                        IF fb_json.HasMember(json_FeederConfigLeft, 'EmptyDelay') THEN
                            json_value := fb_json.FindMember(json_FeederConfigLeft, 'EmptyDelay');
                            PERS.recipeList[i + 0].st120.FeederConfigLeft.EmptyDelay
                                := TO_DINT(fb_json.GetInt(json_value));
                        END_IF
                    END_IF

                    IF fb_json.HasMember(json_st120, 'FeederConfigRight') THEN
                        json_FeederConfigRight := fb_json.FindMember(json_st120, 'FeederConfigRight');

                        IF fb_json.HasMember(json_FeederConfigRight, 'InFilterDelay') THEN
                            json_value := fb_json.FindMember(json_FeederConfigRight, 'InFilterDelay');
                            PERS.recipeList[i + 0].st120.FeederConfigRight.InFilterDelay
                                := TO_DINT(fb_json.GetInt(json_value));
                        END_IF

                        IF fb_json.HasMember(json_FeederConfigRight, 'StartDelay') THEN
                            json_value := fb_json.FindMember(json_FeederConfigRight, 'StartDelay');
                            PERS.recipeList[i + 0].st120.FeederConfigRight.StartDelay
                                := TO_DINT(fb_json.GetInt(json_value));
                        END_IF

                        IF fb_json.HasMember(json_FeederConfigRight, 'StopDelay') THEN
                            json_value := fb_json.FindMember(json_FeederConfigRight, 'StopDelay');
                            PERS.recipeList[i + 0].st120.FeederConfigRight.StopDelay
                                := TO_DINT(fb_json.GetInt(json_value));
                        END_IF

                        IF fb_json.HasMember(json_FeederConfigRight, 'EmptyDelay') THEN
                            json_value := fb_json.FindMember(json_FeederConfigRight, 'EmptyDelay');
                            PERS.recipeList[i + 0].st120.FeederConfigRight.EmptyDelay
                                := TO_DINT(fb_json.GetInt(json_value));
                        END_IF
                    END_IF
                END_IF

                IF fb_json.HasMember(json_i, 'st125') THEN
                    json_st125 := fb_json.FindMember(json_i, 'st125');

                    IF fb_json.HasMember(json_st125, 'xUseVerLeft') THEN
                        json_value := fb_json.FindMember(json_st125, 'xUseVerLeft');
                        PERS.recipeList[i + 0].st125.xUseVerLeft
                            := (fb_json.GetBool(json_value));
                    END_IF

                    IF fb_json.HasMember(json_st125, 'xUseVerRight') THEN
                        json_value := fb_json.FindMember(json_st125, 'xUseVerRight');
                        PERS.recipeList[i + 0].st125.xUseVerRight
                            := (fb_json.GetBool(json_value));
                    END_IF

                    IF fb_json.HasMember(json_st125, 'FeederConfig') THEN
                        json_FeederConfig := fb_json.FindMember(json_st125, 'FeederConfig');

                        IF fb_json.HasMember(json_FeederConfig, 'InFilterDelay') THEN
                            json_value := fb_json.FindMember(json_FeederConfig, 'InFilterDelay');
                            PERS.recipeList[i + 0].st125.FeederConfig.InFilterDelay
                                := TO_DINT(fb_json.GetInt(json_value));
                        END_IF

                        IF fb_json.HasMember(json_FeederConfig, 'StartDelay') THEN
                            json_value := fb_json.FindMember(json_FeederConfig, 'StartDelay');
                            PERS.recipeList[i + 0].st125.FeederConfig.StartDelay
                                := TO_DINT(fb_json.GetInt(json_value));
                        END_IF

                        IF fb_json.HasMember(json_FeederConfig, 'StopDelay') THEN
                            json_value := fb_json.FindMember(json_FeederConfig, 'StopDelay');
                            PERS.recipeList[i + 0].st125.FeederConfig.StopDelay
                                := TO_DINT(fb_json.GetInt(json_value));
                        END_IF

                        IF fb_json.HasMember(json_FeederConfig, 'EmptyDelay') THEN
                            json_value := fb_json.FindMember(json_FeederConfig, 'EmptyDelay');
                            PERS.recipeList[i + 0].st125.FeederConfig.EmptyDelay
                                := TO_DINT(fb_json.GetInt(json_value));
                        END_IF
                    END_IF
                END_IF

                IF fb_json.HasMember(json_i, 'st145') THEN
                    json_st145 := fb_json.FindMember(json_i, 'st145');

                    IF fb_json.HasMember(json_st145, 'xUseVerLeft') THEN
                        json_value := fb_json.FindMember(json_st145, 'xUseVerLeft');
                        PERS.recipeList[i + 0].st145.xUseVerLeft
                            := (fb_json.GetBool(json_value));
                    END_IF

                    IF fb_json.HasMember(json_st145, 'xUseVerRight') THEN
                        json_value := fb_json.FindMember(json_st145, 'xUseVerRight');
                        PERS.recipeList[i + 0].st145.xUseVerRight
                            := (fb_json.GetBool(json_value));
                    END_IF

                    IF fb_json.HasMember(json_st145, 'FeederConfig') THEN
                        json_FeederConfig := fb_json.FindMember(json_st145, 'FeederConfig');

                        IF fb_json.HasMember(json_FeederConfig, 'InFilterDelay') THEN
                            json_value := fb_json.FindMember(json_FeederConfig, 'InFilterDelay');
                            PERS.recipeList[i + 0].st145.FeederConfig.InFilterDelay
                                := TO_DINT(fb_json.GetInt(json_value));
                        END_IF

                        IF fb_json.HasMember(json_FeederConfig, 'StartDelay') THEN
                            json_value := fb_json.FindMember(json_FeederConfig, 'StartDelay');
                            PERS.recipeList[i + 0].st145.FeederConfig.StartDelay
                                := TO_DINT(fb_json.GetInt(json_value));
                        END_IF

                        IF fb_json.HasMember(json_FeederConfig, 'StopDelay') THEN
                            json_value := fb_json.FindMember(json_FeederConfig, 'StopDelay');
                            PERS.recipeList[i + 0].st145.FeederConfig.StopDelay
                                := TO_DINT(fb_json.GetInt(json_value));
                        END_IF

                        IF fb_json.HasMember(json_FeederConfig, 'EmptyDelay') THEN
                            json_value := fb_json.FindMember(json_FeederConfig, 'EmptyDelay');
                            PERS.recipeList[i + 0].st145.FeederConfig.EmptyDelay
                                := TO_DINT(fb_json.GetInt(json_value));
                        END_IF
                    END_IF
                END_IF
            END_IF

            IF fb_json.HasMember(json_i, 'st180') THEN
                json_st180 := fb_json.FindMember(json_i, 'st180');

                IF fb_json.HasMember(json_st180, 'xUseVerLeft') THEN
                    json_value                               := fb_json.FindMember(json_st180, 'xUseVerLeft');
                    PERS.recipeList[i + 0].st180.xUseVerLeft := (fb_json.GetBool(json_value));
                END_IF

                IF fb_json.HasMember(json_st180, 'xUseVerRight') THEN
                    json_value                                := fb_json.FindMember(json_st180, 'xUseVerRight');
                    PERS.recipeList[i + 0].st180.xUseVerRight := (fb_json.GetBool(json_value));
                END_IF
            END_IF
        END_FOR
    END_IF
END_IF

IF fb_json.HasMember(json_head, 'iRecipeCurrent') THEN
    json_value          := fb_json.FindMember(json_head, 'iRecipeCurrent');
    PERS.iRecipeCurrent := TO_INT(fb_json.GetInt(json_value));
END_IF

END_FUNCTION

// ---- POUs/20_AUTO/Mover/DistToTravel.TcPOU
// Get the distance to travel from startPos to stopPos
FUNCTION DistToTravel : LREAL
VAR_INPUT
    startPos : LREAL;
    stopPos  : LREAL;
END_VAR
VAR
END_VAR

IF startPos > stopPos THEN
    DistToTravel := stopPos - startPos + CONST.MAX_TRACK_LENGTH;
ELSE
    DistToTravel := stopPos - startPos;
END_IF

END_FUNCTION

// ---- POUs/20_AUTO/Mover/FB_Group.TcPOU
// Create station group and manage shuttle behaviour 
FUNCTION_BLOCK FB_Group IMPLEMENTS IObject
VAR_INPUT
END_VAR
VAR_OUTPUT
END_VAR
VAR
    _GroupNumber : INT; // group number

    _StationList : ARRAY[1..CONST.MAX_STATION_PER_GROUP] OF POINTER TO FB_Station; // Array of member station member

    _LastVisitedIndex : INT; // Last visited station index
    _MaxStationList   : INT; // The current maximum of station in this group. 0 means no station are present
	
	_iID : INT := 0; // instance ID, is set during FB_Init using the value of _iInstanceCounter 
END_VAR
VAR_STAT
	_iInstanceCounter : INT; // instance counter
END_VAR

METHOD AddStation : REFERENCE TO FB_Group
VAR_INPUT
    station : REFERENCE TO FB_Station;
END_VAR
IF THIS^._MaxStationList < CONST.MAX_STATION_PER_GROUP THEN
    THIS^._MaxStationList                     := THIS^._MaxStationList + 1;
    THIS^._StationList[THIS^._MaxStationList] := ADR(station);
ELSE
    ASSERT(0);
END_IF
END_METHOD

METHOD Equals : BOOL
VAR_INPUT
    object : ANY;
END_VAR
Equals := THIS = object.pValue;
END_METHOD

METHOD FB_init : BOOL
VAR_INPUT
    bInitRetains : BOOL; // if TRUE, the retain variables are initialized (warm start / cold start)
    bInCopyCode  : BOOL; // if TRUE, the instance afterwards gets moved into the copy code (online change)
END_VAR
THIS^._iInstanceCounter := THIS^._iInstanceCounter + 1;
THIS^._iID              := THIS^._iInstanceCounter;

THIS^._MaxStationList   := 0;
THIS^._LastVisitedIndex := 1; // the last station is set to the first

IF THIS^._iID <= CONST.MAX_GROUP THEN
    THIS^._GroupNumber := THIS^._iID;
ELSE
    ASSERT(0);
END_IF
END_METHOD

// The next station is always the one before the last visited
METHOD GetNextStation : REFERENCE TO FB_Station
VAR_INPUT
END_VAR
(* Note about this algorithme :
 * The goal of this algorithm is to divide equaly the use of each station
 * so the wear of station is the same. Other algorithm can be implemented 
 * if needed.
*)
IF THIS^._LastVisitedIndex <= 1 THEN
    THIS^._LastVisitedIndex := THIS^._MaxStationList;
ELSE
    THIS^._LastVisitedIndex := THIS^._LastVisitedIndex - 1;
END_IF

IF THIS^._LastVisitedIndex <= 1 THEN
	ASSERT(0); // we use array of station from 1 to max_station
	THIS^._LastVisitedIndex := 1;
END_IF

GetNextStation REF= THIS^._StationList[THIS^._LastVisitedIndex]^;
END_METHOD

PROPERTY GroupNumber : INT
GET
GroupNumber := this^._GroupNumber;
END_GET
END_PROPERTY

METHOD ToString : STRING
VAR_INPUT
END_VAR
ToString := CONCAT('FB_Station_', TO_STRING(THIS^._iID));
END_METHOD

END_FUNCTION_BLOCK

// ---- POUs/20_AUTO/Mover/FB_StationMan.TcPOU
FUNCTION_BLOCK FB_StationMan IMPLEMENTS IObject
VAR_INPUT
END_VAR
VAR_OUTPUT
END_VAR
VAR
    // a null terminated array of working station
    _WorkStationList : ARRAY[1..CONST.STATION_NUMBER] OF POINTER TO FB_Station;
    _PieceHolder     : REFERENCE TO FB_PieceHolder;

    _GroupList : ARRAY[1..CONST.MAX_GROUP] OF FB_Group;

    _iID : INT := 0; // instance ID, is set during FB_Init using the value of _iInstanceCounter 
END_VAR
VAR_STAT
    _iInstanceCounter : INT := 1; // instance counter
END_VAR

METHOD Equals : BOOL
VAR_INPUT
    object : ANY;
END_VAR
Equals := THIS = object.pValue;
END_METHOD

METHOD FB_init : BOOL
VAR_INPUT
    bInitRetains : BOOL; // if TRUE, the retain variables are initialized (warm start / cold start)
    bInCopyCode  : BOOL; // if TRUE, the instance afterwards gets moved into the copy code (online change)

    // The full station list of the application
    StationList : POINTER TO ARRAY[1..CONST.STATION_NUMBER] OF FB_Station;
    // Used to determine which station is used
    SelStationList : POINTER TO ARRAY[1..CONST.STATION_NUMBER] OF INT;
    PieceHolder    : REFERENCE TO FB_PieceHolder;

END_VAR
VAR
    i                 : INT;
    selStationCounter : INT := 1;
END_VAR
THIS^._iID              := THIS^._iInstanceCounter;
THIS^._iInstanceCounter := THIS^._iInstanceCounter + 1;

FOR i := 1 TO const.STATION_NUMBER BY 1 DO
    IF SelStationList^[i] >= 0 THEN
        THIS^._WorkStationList[selStationCounter] := ADR(StationList^[i]);

        selStationCounter := selStationCounter + 1;
    END_IF
END_FOR

_PieceHolder REF= PieceHolder;
THIS^.SetGroupMembers(StationList, SelStationList);
END_METHOD

// Return the closest station using the station position 
// First we search if we are in range with our set of station
// then, if no station are in our range, we give the nearest next
// station
METHOD PRIVATE FindCloserStationIndex : INT
VAR_INPUT
    CurrentPosition : LREAL;
END_VAR
VAR
    i : INT;
END_VAR
FindCloserStationIndex := -1;

// First we check if we are not in range of a station from our set
FOR i := 1 TO CONST.STATION_NUMBER BY 1 DO
    IF 0 <> THIS^._WorkStationList[i] THEN
        IF THIS^._WorkStationList[i]^.Position.isInPos(CurrentPosition) THEN
            FindCloserStationIndex := i;
            RETURN;
        END_IF
    END_IF
END_FOR

// Then, if no station are in the range, we give the most nearest station, if possible
FOR i := 1 TO CONST.STATION_NUMBER BY 1 DO
    IF 0 <> THIS^._WorkStationList[i] THEN
        IF __ISVALIDREF(THIS^._WorkStationList[i]^.Position) AND
           THIS^._WorkStationList[i]^.Position.lrWorkPosition > CurrentPosition THEN
            FindCloserStationIndex := i;
            EXIT;
        END_IF
    END_IF
END_FOR
END_METHOD

// Return the next station to visit
METHOD GetNextStation : REFERENCE TO FB_Station
VAR_INPUT
    CurrentStation : REFERENCE TO FB_Station;
END_VAR
VAR
    CurrStationIndex : INT;
END_VAR
GetNextStation   REF= CurrentStation;
CurrStationIndex := THIS^.GetStationIndex(CurrentStation);

IF CurrStationIndex > 0 THEN

    IF CurrentStation.GroupNumber > 0 THEN
		// We search for a station which is not from the same group
        WHILE GetNextStation.GroupNumber = CurrentStation.GroupNumber DO
            CurrStationIndex := THIS^.GetNextStationIndex(CurrStationIndex);
            GetNextStation   REF= THIS^._WorkStationList[CurrStationIndex]^;
        END_WHILE
    ELSE
        CurrStationIndex := THIS^.GetNextStationIndex(CurrStationIndex);
        GetNextStation   REF= THIS^._WorkStationList[CurrStationIndex]^;
    END_IF

    // We take a look of the group member and then set the corresponding station
    IF GetNextStation.GroupNumber > 0 THEN
        GetNextStation REF= THIS^._GroupList[GetNextStation.GroupNumber].GetNextStation();
    END_IF

    // when the current is not on the list, we try to move to the nearest
    // but only on the positive direction
ELSE
    CurrStationIndex := THIS^.FindCloserStationIndex(CurrentStation.Position.lrWorkPosition);

    IF CurrStationIndex > 0 THEN
        GetNextStation REF= THIS^._WorkStationList[CurrStationIndex]^;

    ELSE
        GetNextStation REF= THIS^._WorkStationList[1]^;

    END_IF
END_IF
END_METHOD

// Return the next station index in the ring buffer of station
METHOD PRIVATE GetNextStationIndex : INT
VAR_INPUT
	CurrStationIndex : INT;
END_VAR
IF CurrStationIndex >= CONST.STATION_NUMBER THEN
    GetNextStationIndex := 1;

ELSIF THIS^._WorkStationList[CurrStationIndex + 1] = 0 THEN
    GetNextStationIndex := 1;

ELSE
    GetNextStationIndex := CurrStationIndex + 1;
END_IF
END_METHOD

// Get the next station with a valid process. If nothing is found, we 
// simply return to the first station (this should be never the case
// since your machine will be useless...)
METHOD GetNextStationWithProcess : REFERENCE TO FB_Station
VAR_INPUT
    CurrentStation : REFERENCE TO FB_Station;
END_VAR
VAR
    // search station with process algorithme
    iSearchNext        : INT; // incremtal variable used to search in a set of next station
    iTempSearchStation : INT; // incremtal variable used to search in a set of next station
    tempStation        : REFERENCE TO FB_Station;
END_VAR
// If nothing found, we return to the first station
GetNextStationWithProcess REF= THIS^._WorkStationList[1]^;

IF __ISVALIDREF(CurrentStation) THEN
    iSearchNext := 1;

    WHILE iSearchNext < CONST.STATION_NUMBER DO
        tempStation REF= THIS^.GetNextStation(CurrentStation);

        IF __ISVALIDREF(tempStation) AND_THEN __ISVALIDREF(tempStation.Process) THEN
            GetNextStationWithProcess REF= tempStation;
            EXIT;
        END_IF

        iSearchNext := iSearchNext + 1;

    END_WHILE
END_IF
END_METHOD

METHOD GetStartStation : POINTER TO FB_Station
VAR_INPUT
    CurrentPosition : LREAL;
END_VAR
VAR
    CurrStationIndex : INT;
END_VAR
//GetStartStation := THIS^._WorkStationList[1];
CurrStationIndex := THIS^.FindCloserStationIndex(CurrentPosition);

IF CurrStationIndex > 0 THEN
    GetStartStation := THIS^._WorkStationList[CurrStationIndex];

ELSE
    GetStartStation := THIS^._WorkStationList[1];

END_IF
END_METHOD

// return the index of a given station, If the index is -1, no station where found
METHOD PRIVATE GetStationIndex : INT
VAR_INPUT
    Station : REFERENCE TO FB_Station;
END_VAR
VAR
    i : INT;
END_VAR
GetStationIndex := -1;

FOR i := 1 TO CONST.STATION_NUMBER BY 1 DO
    IF Station.Equals(THIS^._WorkStationList[i]^) THEN
        GetStationIndex := i;
        EXIT;
    END_IF
END_FOR
END_METHOD

METHOD IsProcessUsed : BOOL
VAR_INPUT
	process : REFERENCE TO FB_AUT_ABSTRACT;
END_VAR
VAR
	i : INT;
END_VAR
FOR i := 1 TO CONST.STATION_NUMBER BY 1 DO
	IF (0 <> THIS^._WorkStationList[i]) AND_THEN __ISVALIDREF(THIS^._WorkStationList[i]^.Process) THEN
		IF THIS^._WorkStationList[i]^.Process.Equals(process) THEN
			IsProcessUsed := TRUE;
			EXIT; 
		END_IF
	END_IF
END_FOR
END_METHOD

PROPERTY PieceHolder : REFERENCE TO FB_PieceHolder
GET
PieceHolder REF= _PieceHolder;
END_GET
SET
_PieceHolder REF= PieceHolder;
END_SET
END_PROPERTY

METHOD SetGroupMembers : REFERENCE TO FB_Group
VAR_INPUT
    // The full station list of the application
    StationList : POINTER TO ARRAY[1..CONST.STATION_NUMBER] OF FB_Station;
    SelStationList : POINTER TO ARRAY[1..CONST.STATION_NUMBER] OF INT;
END_VAR
VAR
    i : INT;
END_VAR
FOR i := 1 TO CONST.STATION_NUMBER BY 1 DO
    IF SelStationList^[i] > 0 AND SelStationList^[i] <= CONST.MAX_GROUP THEN
        THIS^._GroupList[SelStationList^[i]].AddStation(StationList^[i]);
		StationList^[i].GroupNumber := SelStationList^[i];
    END_IF
END_FOR
END_METHOD

METHOD ToString : STRING
VAR_INPUT
END_VAR
VAR
END_VAR
ToString := CONCAT('FB_StationMan_', TO_STRING(THIS^._iID));
END_METHOD

END_FUNCTION_BLOCK

// ---- POUs/20_AUTO/Simu/FB_Simu_Feeder.TcPOU
// This simu FB is used to generate pieces randomly
// A piece is given during a given amount of time throug 'xOUT_NewPiece'
// Use this output as your nearest sensor 
FUNCTION_BLOCK FB_Simu_Feeder
VAR_INPUT
    xIN_Enable         : BOOL; // enable the feeder
    xIN_PceSensor      : BOOL; // physical piece sensor, when simu_fifo is disabled, xOUT_NewPiece taks this value
    tIN_NewPieceTime   : DINT;
    iIN_WaitTimeMin_ms : DINT;
    iIN_WaitTimeMax_ms : DINT;
END_VAR
VAR_OUTPUT
    xOUT_NewPiece : BOOL;
END_VAR
VAR
    _rand          : DRAND;
    _enableClock   : BOOL  := FALSE;
    _startTime_ms  : UDINT := 0;
    _timeToWait_ms : DINT  := 0;
END_VAR

IF xIN_Enable AND NOT _EnableClock THEN
    THIS^.GetNewRandomTime();
    xOUT_NewPiece := FALSE;
END_IF

_EnableClock := xIN_Enable;

IF xIN_Enable AND THIS^.IsTimeElapsed() THEN
    IF NOT xOUT_NewPiece THEN
        _timeToWait_ms := tIN_NewPieceTime;
		THIS^._startTime_ms := GetTick();
    ELSE
        THIS^.GetNewRandomTime();
    END_IF

    xOUT_NewPiece := NOT xOUT_NewPiece;
ELSIF NOT xIN_Enable THEN
    xOUT_NewPiece := xIN_PceSensor;
END_IF

METHOD FB_init : BOOL
VAR_INPUT
	bInitRetains : BOOL; // if TRUE, the retain variables are initialized (warm start / cold start)
	bInCopyCode : BOOL;  // if TRUE, the instance afterwards gets moved into the copy code (online change)
END_VAR
VAR
END_VAR
this^._rand.Seed := TO_INT(F_GetSystemTime());
END_METHOD

METHOD PRIVATE GetNewRandomTime : BOOL
VAR_INPUT
END_VAR
THIS^._startTime_ms := GetTick();
THIS^._rand();
THIS^._timeToWait_ms :=
    TO_DINT(THIS^._rand.Num * (THIS^.iIN_WaitTimeMax_ms - THIS^.iIN_WaitTimeMin_ms) + THIS^.iIN_WaitTimeMin_ms);
END_METHOD

METHOD IsTimeElapsed : BOOL
VAR_INPUT
END_VAR
IsTimeElapsed := TO_DINT(GetTick() - _startTime_ms) > _timeToWait_ms;
END_METHOD

END_FUNCTION_BLOCK

// ---- POUs/20_AUTO/ST100/FB_AUT_LOAD.TcPOU
FUNCTION_BLOCK FB_AUT_LOAD EXTENDS FB_AUT_ABSTRACT IMPLEMENTS ISimuMoverTimers
    (****************************************************************************)
    (*	POU_AUT_zxx			Bausteinaufrufe Station	zxx							*)
    (*	Status				ungetestet											*)
    (*  Version:			1.0													*)
    (*	Beschrieb:																*)
    (*																			*)
    (*	Abläufe:			FB_ABLzxxA		Hauptablauf							*)
    (*																			*)
    (*																			*)
    (* 	25.09.2019/Dj															*)
    (****************************************************************************)
    (*	dd.mm.yyyy   KZ    x.y			Beschrieb								*)
    (****************************************************************************)
VAR_INPUT
    (* spezifische Eingänge *)

END_VAR
VAR_OUTPUT
    (* spezifische Ausgänge *)

END_VAR
VAR
    (* Bausteine *)
    _FB_ABL_100A : FB_ABL_LOAD;
END_VAR

(*******************************************************************)
(* Timer *)
(*******************************************************************)

(*******************************************************************)
(* Flanken / Merker *)
(*******************************************************************)
//MANU CYCLE
IF (enIN_State = StateMANU) AND xIN_ManuCycle THEN
    xManuCycle := TRUE;
END_IF;

IF (enIN_State <> StateMANU) OR xOUT_Done THEN
    xManuCycle := FALSE;
END_IF

//NEXT STEP
xNextStep := (enIN_State > StateSTEP) OR
             ((enIN_State = StateSTEP) AND xIN_Step) OR
             ((enIN_State = StateMANU) AND xManuCycle);

//RESET
xReset := (enIN_State < StateREADY) AND (enIN_State <> StateINIT) AND NOT xManuCycle;

(*******************************************************************)
(* Bausteinaufrufe Abläufe *)
(*******************************************************************)

_FB_ABL_100A(xIN_Reset    := xReset,
             xIN_Init     := xIN_Init,
             xIN_Quit     := xIN_Quit,
             xIN_Start    := enIN_State = enState.StateAUTO, //AND _FB_ABL_100A.xOUT_Done AND _FB_ABL_100A.xOUT_Ready,
             xIN_Sperre   := NOT xIN_On,
             xIN_NextStep := xNextStep,
             xIN_AlarmAktiv
                 := xIN_AlarmAktiv,
             xIN_DryCycle    := xIN_DryCycle,
             xIN_RestartCYCL := enIN_State = enState.StateAUTO, // only restart when the mover has move out
             enIN_State      := enIN_State,
             tIN_Timeout     := tIN_Timeout,
             pxFG_Freigabe   := ADR(xRelease),
             Mover           := THIS^.Mover,
             xOUT_ErrFlag    =>,
             xOUT_Busy       =>,
             xOUT_Done       =>,
             xOUT_Timeout    =>,
             xOUT_InitDone   =>,
             xOUT_Wait       =>,
             iOUT_Step       =>,
             bOUT_Error      =>);

(*******************************************************************)
(* Mover reset flags *)
(*******************************************************************)

(*******************************************************************)
(* OUTPUT *)
(*******************************************************************)
xOUT_InitDone := _FB_ABL_100A.xOUT_InitDone;
xOUT_Ready    := xOUT_InitDone;
xOUT_Done     := _FB_ABL_100A.xOUT_Done;
xOUT_ErrFlag  := _FB_ABL_100A.xOUT_ErrFlag;
xOUT_Wait     := _FB_ABL_100A.xOUT_Wait;
xOUT_AlarmST  := xOUT_ErrFlag;

(*******************************************************************)
(* Bausteinaufruf Error Station *)
(*******************************************************************)
// POU_ERR_VORLAGE(xIN_QUIT:=xIN_Quit , pstrArIN_ALARM:=ADR(HMI.strArALARM[1]));

METHOD GiveMover : IProcessSampleMover
VAR_INPUT
	mover : REFERENCE TO FB_Mover;
END_VAR
IF __ISVALIDREF(mover) THEN
    THIS^.Mover                       REF= mover;
END_IF
END_METHOD

(* % of completion of the process *)
PROPERTY iCompletionPC : INT
GET
iCompletionPC := THIS^._FB_ABL_100A.iOUT_ProcessCompletion;
END_GET
END_PROPERTY

(* Process time, expressed in milisecond *)
PROPERTY iProcessTimeMili_1 : DINT
GET
iProcessTimeMili_1 := TO_DINT(this^._FB_ABL_100A.iProcessTimeMili1);
END_GET
SET
THIS^._FB_ABL_100A.iProcessTimeMili1 := TO_UDINT(iProcessTimeMili_1);
END_SET
END_PROPERTY

(* Process time, expressed in milisecond *)
PROPERTY iProcessTimeMili_2 : DINT
GET
iProcessTimeMili_2 := TO_DINT(this^._FB_ABL_100A.iProcessTimeMili2);
END_GET
SET
THIS^._FB_ABL_100A.iProcessTimeMili2 := TO_UDINT(iProcessTimeMili_2);
END_SET
END_PROPERTY

PROPERTY ProcessExecution : ProcessExecution_e
GET
ProcessExecution := THIS^._ProcessExecution;
END_GET
SET
THIS^._ProcessExecution := ProcessExecution;
END_SET
END_PROPERTY

METHOD TakeMover : IProcessSampleMover
VAR_INPUT
END_VAR
THIS^.Mover REF= 0;
END_METHOD

PROPERTY xBusy : BOOL
GET
xBusy := This^._FB_ABL_100A.xOUT_Busy;
END_GET
SET
END_SET
END_PROPERTY

PROPERTY xDone : BOOL
GET
xDone := THIS^._FB_ABL_100A.xOUT_Ready OR THIS^._FB_ABL_100A.xOUT_Done;
END_GET
END_PROPERTY

PROPERTY xMoverPathFree : BOOL
GET
xMoverPathFree := THIS^._FB_ABL_100A.xOUT_MoverFree OR THIS^._FB_ABL_100A.xOUT_Ready OR THIS^._FB_ABL_100A.xOUT_Done;
END_GET
END_PROPERTY

PROPERTY xMoverShouldLeave : BOOL
GET
xMoverShouldLeave := THIS^._FB_ABL_100A.iOUT_Step = ST100_Load_e.SYNC_MOVER_LEAVE;
END_GET
END_PROPERTY

END_FUNCTION_BLOCK

// ---- POUs/20_AUTO/ST105/FB_ABL_105_Pnp.TcPOU
FUNCTION_BLOCK FB_ABL_105_Pnp
(****************************************************************************************)
(*	TITEL				RFID-Ring laden		    										*)
(*	Status				ungetestet                         								*)
(*	Beschrieb:			Ablaufbeschreibung												*)
(*																						*)
(*	Steps:	self-explained using enum													*)
(***********************************Revisionen*******************************************)
(*	see github blames																	*)
(****************************************************************************************)

VAR_INPUT
    xIN_Reset       : BOOL;          // Schrittkette zurücksetzen 
    xIN_Init        : BOOL;          // Initialisieren
    xIN_Quit        : BOOL;          // Fehler quittieren 
    xIN_Start       : BOOL;          // Startbefehl
    xIN_Sperre      : BOOL;          // FB Sperren 
    xIN_NextStep    : BOOL;          // Nächsten Schritt ausführen 
    xIN_AlarmAktiv  : BOOL;          // Anlage hat Alarm
    xIN_DryCycle    : BOOL;          // Fahren ohne Teile
    xIN_RestartCYCL : BOOL;          // Zyklus erneut starten im STEP, END, LEERFAHREN
    enIN_State      : enState;       // Status Anlage
    tIN_Timeout     : TIME := T#10s; // Timout

    pxFG_Freigabe : POINTER TO BOOL; //Freigabe von Station

    // Application specific
    Mover              : REFERENCE TO FB_Mover;
    xIN_PceReadyToPick : BOOL; // the piece(s) is/are ready to picked
END_VAR
VAR_OUTPUT
    (* standart Ausgänge *)
    xOUT_ErrFlag  : BOOL;        // Error Flag 
    xOUT_Busy     : BOOL;        // Baustein befindet sich im Ablauf 
    xOUT_Done     : BOOL;        // Baustein hat den Ablauf beendet 		
    xOUT_Ready    : BOOL;        // Ready to begin, should be the same state as done	
    xOUT_Timeout  : BOOL;        // Timeout FB 
    xOUT_InitDone : BOOL;        // initialisierung fertig
    xOUT_Wait     : BOOL;        // Wartet auf Bedingung
    iOUT_Step     : ST105_Pnp_e; // Aktueller Schritt 
    sOUT_Step     : STRING;      // Aktueller Schritt but in string format
    bOUT_Error    : BYTE;        // Fehlernummer

    iOUT_ProcessCompletion : INT;  //process completion, express in % (0-100)
    xOUT_MoverFree         : BOOL; // The mover is free to move
    xOUT_PickPiece         : BOOL; // Set to true when a piece is picked

END_VAR
VAR
    (* Standard *)
    (* Schritt *)
    iLastStep : ST105_Pnp_e; // Merker letzter Schritt 
    iPreStep  : ST105_Pnp_e; // Schritt zurück nach Alarm 
    iAktStep  : ST105_Pnp_e; // aktueller Schritt

    // Trigger Starten 
    rtSTART : R_TRIG;
    // Timer TimeOut 
    TON_Timeout : TON;

    (* Bausteine *)

    (* Spezial *)
    fb_axis105_11Z : FB_AxisLM_V1_1;

    fb_PnpVerAxisU : FB_LinearMotionMan;

    fb_simu_axis105_11Z : FB_Simu_AxisLM_V1_1;

    fanuc_cmd    AT %Q* : Fanuc_hw_command_to_robot_t;
    fanuc_status AT %I* : Fanuc_status_std_from_robot;

    aut_cmd_to_robot      AT %Q* : ST105_Fanuc_command_t;
    aut_status_from_robot AT %I* : ST105_Fanuc_status_t;

    PickOffset_X_deci AT %Q* : UINT; // X offset of picking position
    PickOffset_Y_deci AT %Q* : UINT; // Y offset of picking position
    PickUpPos_Z_deci  AT %Q* : UINT; // Z traveling height from pick to place position

    hmi_force_place    : BOOL;
    hmi_force_in_place : BOOL;

END_VAR
VAR CONSTANT
    PNP_SIMULATION : BOOL := FALSE; // Set to TRUE to simulate this part of the program
END_VAR

(*******************************************************************)
(* Trigger  *)
(*******************************************************************)
(* Zurücksetzen *)
IF xIN_RESET THEN
    iPreStep  := ST105_Pnp_e.RESET;
    iOUT_Step := ST105_Pnp_e.RESET;
END_IF;

(* Error Quittieren *)
IF (bOUT_Error <> 0) AND xIN_Quit THEN
    xOUT_ErrFlag := FALSE;
    bOUT_Error   := 0;
    iOUT_Step    := iPreStep;
END_IF;

(*******************************************************************)
(* Timer *)
(*******************************************************************)
TON_Timeout(IN := xIN_NextStep AND (iLastStep = iOUT_Step) (*todo FG *) ,
            PT := tIN_Timeout);

(*******************************************************************)
(* Bausteine *)
(*******************************************************************)
fb_PnpVerAxisU(config          := _20_AUTO.recipe.linearAxis[LinearAxis_e.ST105_11Z],
               xIN_Init        := enIN_State = enState.StateINIT,
               xIN_Reset       := xIN_Reset,
               lrIN_CurrPos    := fb_axis105_11Z.rOUT_ActPos,
               lrIN_Delta_mm   := 0.5,
               iIN_CurrentStep := iOUT_Step,
               iIN_moveNumber  := ST105_PnpVerPushPos_e._max);

fb_simu_axis105_11Z(xIN_Enable          := PNP_SIMULATION AND CONST.USE_SIMULATION,
                    bIN_AxisCntr        := fb_axis105_11Z.bOUT_AxisCntr,
                    wIN_AxisState       := ST105_Axis.axis105_11Z.wState,
                    udiIN_HomingTime_ms := 2000,
                    pIN_axisSimu        := ADR(SIMU.axis_ref[Axis_e.ST105_11Z]),
                    pIN_axisHW          := ADR(ST105_Axis.axis105_11Z.axis),
                    rIN_PosActual       := ST105_Axis.axis105_11Z.rActPos,
                    rIN_PosMax          := ST105_Axis.const105_11Z.POS_MAX,
                    rIN_PosMin          := ST105_Axis.const105_11Z.POS_MIN,
                    rIN_PixMax          := 100,
                    rIN_PixMin          := 0);

fb_axis105_11Z(enIN_State       := enIN_State,
               parIN_Buttons    := ADR(AXIS.btTeachArAxis[Axis_e.ST105_11Z]),
               xIN_DisButtons   := FALSE,
               xIN_Quit         := xIN_Quit,
               xIN_PARAMok      := TRUE,
               xIN_FREE         := TRUE,
               xIN_FREE_HOME    := TRUE,
               rIN_POSMIN       := ST185_Axis.const185_10Z.POS_MIN,
               rIN_POSMAX       := ST185_Axis.const185_10Z.POS_MAX,
               rIN_VELOMAX      := ST185_Axis.const185_10Z.VELO_MAX,
               rIN_VELOMANU     := ST185_Axis.const185_10Z.VELO_MANU,
               rIN_VELOOPEN     := ST185_Axis.const185_10Z.POS_MAX / 4,
               rIN_JogInc       := AXIS.rTeachIncAxis,
               xIN_Execute      := fb_PnpVerAxisU.xOUT_Execute,
               xIN_Relative     :=,
               xIN_STOP         :=,
               xIN_OFF          :=,
               rIN_Position     := TO_REAL(fb_PnpVerAxisU.OUT_MoveProfile.lrPosition),
               rIN_Velocity     := TO_REAL(fb_PnpVerAxisU.OUT_MoveProfile.lrVelocity),
               rIN_Acceleration := TO_REAL(fb_PnpVerAxisU.OUT_MoveProfile.lrAccel),
               rIN_Deceleration := TO_REAL(fb_PnpVerAxisU.OUT_MoveProfile.lrDecel),
               rIN_Jerk         := TO_REAL(fb_PnpVerAxisU.OUT_MoveProfile.lrJerk),
               rIN_PosManu      := TO_REAL(_20_AUTO.recipe.linearAxis[LinearAxis_e.ST105_11Z]
                                               .movesList[AXIS.bTeachPos[Axis_e.ST105_11Z]].lrPosition),
               rIN_VeloJogManu := TO_REAL(Axis.rJogVelo_pc),
               xIN_Home        := ST105_Pnp_e.Init_HomeVertical = iOUT_Step,
               xIN_Reset       := (ST105_Pnp_e.RESET = iOUT_Step) OR xIN_Reset,
               wAxisState      := fb_simu_axis105_11Z.wOUT_AxisState,
               bOUT_AxisCntr   => ST105_Axis.axis105_11Z.bCtrlHi,
               rOUT_ActPos     => ST105_Axis.axis105_11Z.rActPos,
               axisIN_REF      := fb_simu_axis105_11Z.pOUT_axisRef^);

(*******************************************************************)
(* OUTPUTS *)
(*******************************************************************)
// Error Flag 
xOUT_ErrFlag := (bOUT_Error <> 0) OR (ST105_Pnp_e.ERROR = iOUT_Step);
// Baustein befindet sich im Ablauf 
xOUT_Busy := (iOUT_Step > ST105_Pnp_e.READY) AND (iOUT_Step < ST105_Pnp_e.DONE);
// Baustein hat den Ablauf beendet
xOUT_Done := (iOUT_Step = ST105_Pnp_e.DONE);
// Process ready
xOUT_Ready := (iOUT_Step = ST105_Pnp_e.READY) OR (iOUT_Step = ST105_Pnp_e.waitOnMover);
// Timeout FB 				 		
xOUT_Timeout := TON_Timeout.Q;
// Itialisierung fertig			
xOUT_InitDone := (iOUT_Step = ST105_Pnp_e.READY) OR (iOUT_Step = ST105_Pnp_e.waitOnMover);
// Aktueller Schritt			
iOUT_Step := iOUT_Step; //Im Ablauf gesetzt		
sOUT_Step := TO_STRING(iOUT_Step);
//Fehlernummer	 
bOUT_Error := bOUT_Error; //Im Ablauf/FB gesetzt	
(* Warte (alle Schritte wo auf FG oder Teile gewartet wird) *)
xOUT_Wait := (iOUT_Step = ST105_Pnp_e.DONE) OR
             (iOUT_Step = ST105_Pnp_e.READY) OR
             (iOUT_Step = ST105_Pnp_e.START) OR
             (iOUT_Step = ST105_Pnp_e.waitOnMover) OR
             (iOUT_Step = ST105_Pnp_e.SYNC_MOVER_LEAVE) OR
             (iOUT_Step = ST105_Pnp_e.wait_on_feeder);

xOUT_MoverFree := iOUT_Step >= ST105_Pnp_e.MOVER_FREE_OP AND iOUT_Step < ST105_Pnp_e.MOVER_NEEDED_OP;

iOUT_ProcessCompletion := F_GetPercent_2(iOUT_Step,
                                         ST105_Pnp_e.wait_on_feeder,
                                         ST105_Pnp_e.pusher_down,
                                         ST105_Pnp_e.Robot_place,
                                         ST105_Pnp_e.pusher_down);

xOUT_PickPiece := iOUT_Step = ST105_Pnp_e.pusher_down;

fanuc_cmd.command_std.IMDSTP     := TRUE AND NOT (PNP_SIMULATION AND CONST.USE_SIMULATION);
fanuc_cmd.command_std.Hold       := TRUE AND NOT (PNP_SIMULATION AND CONST.USE_SIMULATION);
fanuc_cmd.command_std.SFSPD      := TRUE AND NOT (PNP_SIMULATION AND CONST.USE_SIMULATION);
fanuc_cmd.command_std.FaultReset := xIN_Quit;
fanuc_cmd.command_std.Start      := iOUT_Step = ST105_Pnp_e.Init_RobotRaiseStartFlag AND
                                    NOT (PNP_SIMULATION AND CONST.USE_SIMULATION);

fanuc_cmd.command_std.Enable := TRUE AND NOT (PNP_SIMULATION AND CONST.USE_SIMULATION);

PickOffset_X_deci := _20_AUTO.recipe.st105.PickOffset_X_deci;
PickOffset_Y_deci := _20_AUTO.recipe.st105.PickOffset_Y_deci;
// add a constant to adjust the screw height of the rotative table
PickUpPos_Z_deci := _20_AUTO.recipe.st105.PickUpPos_Z_deci + UINT#500;

aut_cmd_to_robot.FG_Pick  := (ST105_Pnp_e.Robot_Pick = iOUT_Step) AND NOT (PNP_SIMULATION AND CONST.USE_SIMULATION);
aut_cmd_to_robot.FG_Place :=
    ((ST105_Pnp_e.Robot_place = iOUT_Step) OR hmi_force_place) AND NOT (PNP_SIMULATION AND CONST.USE_SIMULATION);

aut_cmd_to_robot.Use_griper_left  := _20_AUTO.recipe.st105.xUseVerLeft;
aut_cmd_to_robot.Use_griper_right := _20_AUTO.recipe.st105.xUseVerRight;

aut_cmd_to_robot.XOff := _20_AUTO.recipe.st105.isPickOffset_X_neg;
aut_cmd_to_robot.YOff := _20_AUTO.recipe.st105.isPickOffset_Y_neg;
aut_cmd_to_robot.ZOff := _20_AUTO.recipe.st105.isPickUpPos_Z_neg;

(*******************************************************************)
(* Ablauf *)
(*******************************************************************)

(* Sperren *)
IF xIN_Sperre THEN
    iPreStep  := ST105_Pnp_e.RESET;
    iOUT_Step := ST105_Pnp_e.RESET;
    RETURN;
END_IF;

(* Schritt Merker *)
IF iAktStep <> iOUT_Step THEN
    iLastStep := iAktStep;
    iAktStep  := iOUT_Step;
END_IF

(* START *)
rtSTART(CLK := xIN_Start);

(*******************************************************************)
(* Schrittkette  *)
(*******************************************************************)
CASE iOUT_Step OF

(***** RESET *****)
ST105_Pnp_e.RESET: (* Schritt 0-99 *)
    //Initialisierungen
    //Start Init Ablauf
    IF xIN_Init THEN
        iOUT_Step := ST105_Pnp_e.INIT;
        //Start Manu Ablauf
    ELSIF enIN_State = StateMANU AND xIN_NextStep THEN
        iOUT_Step := ST105_Pnp_e.INIT;
    END_IF;

(***** INIT *****)
ST105_Pnp_e.INIT: (* Grundstellung ? *)
    IF fb_axis105_11Z.xOUT_HOMED THEN
        iOUT_Step := ST105_Pnp_e.Init_VerticalDown;
    ELSE
        iOUT_Step := ST105_Pnp_e.Init_HomeVertical;
    END_IF

ST105_Pnp_e.Init_HomeVertical:
    IF fb_axis105_11Z.xOUT_HOMED THEN
        iOUT_Step := ST105_Pnp_e.Init_VerticalDown;
    END_IF

ST105_Pnp_e.Init_VerticalDown:
    IF fb_PnpVerAxisU.MoveTo(ST105_PnpVerPushPos_e.down).xOUT_InPos THEN
        IF fanuc_status.PRG_Running THEN
            iOUT_Step := ST105_Pnp_e.Init_check_if_pces_handled;
        ELSE
            iOUT_Step := ST105_Pnp_e.Init_RobotRaiseStartFlag;
        END_IF
    END_IF

ST105_Pnp_e.Init_RobotRaiseStartFlag:
    IF TRUE THEN // maybe a tempo or a flag from the robot is needed here
        iOUT_Step := ST105_Pnp_e.Init_check_if_pces_handled;
    END_IF

ST105_Pnp_e.Init_RobotFallStartFlag:
    IF fanuc_status.PRG_Running OR (PNP_SIMULATION AND CONST.USE_SIMULATION) THEN
        iOUT_Step := ST105_Pnp_e.Init_check_if_pces_handled;
    END_IF

ST105_Pnp_e.Init_check_if_pces_handled:
    IF TRUE THEN
        IF aut_status_from_robot.Ready_to_place THEN
            iOUT_Step := ST105_Pnp_e.waitOnMover;
        ELSE
            iOUT_Step := ST105_Pnp_e.READY;
        END_IF
    END_IF

(***** READY / INIT DONE *****)
ST105_Pnp_e.READY:    (* Start AUTO,END,LEER,STEP *)
    IF xIN_Start THEN //IF rtSTART.Q THEN
        iOUT_Step := ST105_Pnp_e.START;
    END_IF

(***** START  ZYKLISCH *****)
ST105_Pnp_e.START: (*  *)
    IF xIN_NextStep AND pxFG_Freigabe^ THEN
        IF enState.StateLEER = enIN_State THEN
            IF aut_status_from_robot.Ready_to_place THEN
                iOUT_Step := ST105_Pnp_e.waitOnMover;
            ELSIF __ISVALIDREF(Mover) THEN
                iOUT_Step := ST105_Pnp_e.SYNC_MOVER_LEAVE;
            END_IF
        ELSE
            iOUT_Step := ST105_Pnp_e.wait_on_feeder;
        END_IF
    END_IF;

ST105_Pnp_e.wait_on_feeder:
    IF xIN_NextStep AND xIN_PceReadyToPick THEN
        iOUT_Step := ST105_Pnp_e.push_up_casing;
    END_IF

ST105_Pnp_e.push_up_casing:
    IF xIN_NextStep AND fb_PnpVerAxisU.MoveTo(ST105_PnpVerPushPos_e.up).xOUT_InPos THEN
        IF PNP_SIMULATION AND CONST.USE_SIMULATION THEN
            IF fb_axis105_11Z.xOUT_DONE THEN // needed beacause we perform 2 movements one after the other
                iOUT_Step := ST105_Pnp_e.pusher_down;
            END_IF
        ELSE
            iOUT_Step := ST105_Pnp_e.Robot_Pick;
        END_IF
    END_IF

ST105_Pnp_e.Robot_Pick:
    IF aut_status_from_robot.Picked THEN
        iOUT_Step := ST105_Pnp_e.Robot_wait_picked_falling;

        // we don't generate an error here since this may hapen
        // when we stop the machine during the robot movement
    ELSIF aut_status_from_robot.Ready_to_place THEN
        iOUT_Step := ST105_Pnp_e.waitOnMover;

    END_IF

ST105_Pnp_e.Robot_wait_picked_falling:
    IF xIN_NextStep AND NOT aut_status_from_robot.Picked THEN
        iOUT_Step := ST105_Pnp_e.pusher_down;
    END_IF

ST105_Pnp_e.pusher_down:
    IF xIN_NextStep AND fb_PnpVerAxisU.MoveTo(ST105_PnpVerPushPos_e.down).xOUT_InPos THEN
        iOUT_Step := ST105_Pnp_e.waitOnMover;
    END_IF

ST105_Pnp_e.waitOnMover: (*  *)
    IF xIN_NextStep AND (__ISVALIDREF(Mover) OR HMI.bArForceCyclusState[StationList_e.ST105]) THEN
        IF (PNP_SIMULATION AND CONST.USE_SIMULATION) OR
           ((enState.StateLEER = enIN_State) AND NOT aut_status_from_robot.Ready_to_place) THEN
            iOUT_Step := ST105_Pnp_e.SYNC_MOVER_LEAVE;
        ELSE
            IF Mover.GetLastStationDone() >= INT#105 THEN
                iOUT_Step := ST105_Pnp_e.SYNC_MOVER_LEAVE;
            ELSE
                iOUT_Step := ST105_Pnp_e.Robot_place;
            END_IF
        END_IF
    END_IF;

ST105_Pnp_e.Robot_place:
    IF aut_status_from_robot.Placed THEN
        iOUT_Step := ST105_Pnp_e.Robot_wait_placed_falling;

        IF __ISVALIDREF(Mover) THEN
            IF NOT Mover.SetLastStation(105) THEN
                ASSERT(0);
            END_IF
        END_IF

        // we don't generate an error here since this may hapen
        // when we stop the machine during the robot movement
    ELSIF aut_status_from_robot.Ready_to_pick THEN
        iOUT_Step := ST105_Pnp_e.wait_on_feeder;

    END_IF

ST105_Pnp_e.Robot_wait_placed_falling:
    IF xIN_NextStep AND NOT aut_status_from_robot.Placed THEN
        iOUT_Step := ST105_Pnp_e.SYNC_MOVER_LEAVE;

        IF __ISVALIDREF(Mover) THEN
            IF NOT Mover.SetLastStation(105) THEN
                ASSERT(0);
            END_IF
        END_IF
    END_IF

ST105_Pnp_e.SYNC_MOVER_LEAVE:
    // The mover needs to be taken by MoverMan
    IF NOT __ISVALIDREF(Mover) THEN
        IF NOT aut_status_from_robot.Ready_to_place THEN
            iOUT_Step := ST105_Pnp_e.DONE;
        ELSE
            iOUT_Step := ST105_Pnp_e.waitOnMover;
        END_IF
    END_IF

(***** DONE *****)
ST105_Pnp_e.DONE: (* Letzter Schritt  *)
    IF NOT xIN_AlarmAktiv THEN
        //AUTO
        IF (enIN_State = StateAUTO) AND xIN_RestartCYCL THEN
            iOUT_Step := ST105_Pnp_e.START;
            //STEP / END / LEERFAHREN restart
        ELSIF (enIN_State < StateAUTO) AND (enIN_State >= enState.StateSTEP) AND xIN_RestartCYCL THEN
            iOUT_Step := ST105_Pnp_e.START;
            //STEP / END / LEERFAHREN fertig
        ELSIF (enIN_State = StateREADY) THEN
            iOUT_Step := ST105_Pnp_e.READY;
        END_IF;
    END_IF;

(************ ERROR *************)
ST105_Pnp_e.ERROR: (* ERROR *) ;

END_CASE;

END_FUNCTION_BLOCK

// ---- POUs/20_AUTO/ST120/FB_ABL_120_Feeder.TcPOU
FUNCTION_BLOCK FB_ABL_120_Feeder
(****************************************************************************************)
(*	TITEL				laden Kristall modul, Feeder and rotary table                   *)
(*	Status				ungetestet                         								*)
(*	Beschrieb:			Ablaufbeschreibung												*)
(*																						*)
(*	Steps:	self-explained using enum													*)
(***********************************Revisionen*******************************************)
(*	see github blames																	*)
(****************************************************************************************)

VAR_INPUT
    xIN_Reset       : BOOL;          // Schrittkette zurücksetzen 
    xIN_Init        : BOOL;          // Initialisieren
    xIN_Quit        : BOOL;          // Fehler quittieren 
    xIN_Start       : BOOL;          // Startbefehl
    xIN_Sperre      : BOOL;          // FB Sperren 
    xIN_NextStep    : BOOL;          // Nächsten Schritt ausführen 
    xIN_AlarmAktiv  : BOOL;          // Anlage hat Alarm
    xIN_DryCycle    : BOOL;          // Fahren ohne Teile
    xIN_RestartCYCL : BOOL;          // Zyklus erneut starten im STEP, END, LEERFAHREN
    enIN_State      : enState;       // Status Anlage
    tIN_Timeout     : TIME := T#10s; // Timout

    pxFG_Freigabe : POINTER TO BOOL; //Freigabe von Station

    // Application specific
    xIN_PickPiece : BOOL; (* signal from the pick and place element
                             the number of picked signal depend on the recipe *)
    xIN_PnpGripperOpen : BOOL; // the gripper of the pnp part is open
    xIN_PnpNotOnTheWay : BOOL; // the pnp is at the track side or up enough
END_VAR
VAR_OUTPUT
    (* standart Ausgänge *)
    xOUT_ErrFlag  : BOOL;           // Error Flag 
    xOUT_Busy     : BOOL;           // Baustein befindet sich im Ablauf 
    xOUT_Done     : BOOL;           // Baustein hat den Ablauf beendet 		
    xOUT_Ready    : BOOL;           // Ready to begin, should be the same state as done	
    xOUT_Timeout  : BOOL;           // Timeout FB 
    xOUT_InitDone : BOOL;           // initialisierung fertig
    xOUT_Wait     : BOOL;           // Wartet auf Bedingung
    iOUT_Step     : ST120_Feeder_e; // Aktueller Schritt 
    sOUT_Step     : STRING;         // Aktueller Schritt but in string format
    bOUT_Error    : BYTE;           // Fehlernummer

    // Application specific
    xOUT_PceReadyToPick : BOOL; // the piece(s) is/are ready to picked
END_VAR
VAR
    (* Standard *)
    (* Schritt *)
    iLastStep : ST120_Feeder_e; // Merker letzter Schritt 
    iPreStep  : ST120_Feeder_e; // Schritt zurück nach Alarm 
    iAktStep  : ST120_Feeder_e; // aktueller Schritt

    // Trigger Starten 
    rtSTART : R_TRIG;
    // Timer TimeOut 
    TON_Timeout : TON;

    (* Bausteine *)
	btfb_feederLeft					: FB_BUTTON;
	btfb_feederRight				: FB_BUTTON;

    // Application specific^
    fb_pivotLeft    : FB_ZylMo2El_V2_1;
    fb_pivotRight   : FB_ZylMo2El_V2_1;
    simu_pivotLeft  : FB_Simu_Zyl2Pos;
    simu_pivotRight : FB_Simu_Zyl2Pos;

    simu_feederLeft  : FB_Simu_Feeder;                    // simulation of a feeder
    simu_feederRight : FB_Simu_Feeder;                    // simulation of a feeder
    simu_fifoLeft    : FB_Fifo(BAND_SIZE_FOR_TUBE_LEFT);  // fifo to hold a piece
    simu_fifoRight   : FB_Fifo(BAND_SIZE_FOR_TUBE_RIGHT); // fifo to hold a piece
    rtPutPieceLeft   : R_TRIG;                            // trigger to add a piece
    rtPutPieceRight  : R_TRIG;                            // trigger to add a piece

    fb_feederLeft      : FB_Feeder2Sensors;
    fb_feederRight     : FB_Feeder2Sensors;
    fb_hubladerLeft    : FB_ZylMo2El_V2_1;
    fb_hubladerRight   : FB_ZylMo2El_V2_1;
    simu_hubladerLeft  : FB_Simu_Zyl2Pos;
    simu_hubladerRight : FB_Simu_Zyl2Pos;

    simu_start_tick : UDINT; // simulation start tick, used to simulate movement

    TON_PieceInPivotLeft  : TON;
    TON_PieceInPivotRight : TON;

END_VAR
VAR CONSTANT
    BAND_SIZE_FOR_TUBE_LEFT  : INT := 3; // Band size, we assume that tubes pushe each other in order to move to the PNP machine
    BAND_SIZE_FOR_TUBE_RIGHT : INT := 2; // Band size, we assume that tubes pushe each other in order to move to the PNP machine

    FEEDER_SIMULATION : BOOL := FALSE; // Simulate this code
END_VAR

(*******************************************************************)
(* Trigger  *)
(*******************************************************************)
(* Zurücksetzen *)
IF xIN_RESET THEN
    iPreStep  := ST120_Feeder_e.RESET;
    iOUT_Step := ST120_Feeder_e.RESET;
END_IF;

(* Error Quittieren *)
IF (bOUT_Error <> 0) AND xIN_Quit THEN
    xOUT_ErrFlag := FALSE;
    bOUT_Error   := 0;
    iOUT_Step    := iPreStep;
END_IF;

(*******************************************************************)
(* Timer *)
(*******************************************************************)
TON_Timeout(IN := xIN_NextStep AND (iLastStep = iOUT_Step) (*todo FG *) ,
            PT := tIN_Timeout);

TON_PieceInPivotLeft(IN := IO_BOX.I6404_ST120_teil_in_vereizelung_links,
                     PT := DINT_TO_TIME(_20_AUTO.recipe.st120.TON_PieceInSeperatorLeft));

TON_PieceInPivotRight(IN := IO_BOX.I6405_ST120_teil_in_vereinzelung_rechts,
                      PT := DINT_TO_TIME(_20_AUTO.recipe.st120.TON_PieceInSeperatorRight));

(*******************************************************************)
(* Bausteine *)
(*******************************************************************)
fb_pivotLeft(xIN_Reset    := xIN_Reset OR (ST120_Feeder_e.RESET = iOUT_Step),
             xIN_Quit     := xIN_Quit,
             xIN_Manu     := enState.StateMANU = enIN_State,
             pbtIN_Button := ADR(HMI.btManuCylinders[StationList_e.ST120][3]),
             xIN_GS       := simu_pivotLeft.xOUT_inGS,
             xIN_AS       := simu_pivotLeft.xOUT_inAS,
             xIN_FREE     := xIN_PnpNotOnTheWay OR xIN_PnpGripperOpen,
             xINtoGS      :=
                 _20_AUTO.recipe.st120.xUseVerLeft AND
                 ((ST120_Feeder_e.rotate_to_pnp = iOUT_Step) OR (ST120_Feeder_e.Init_pivot_to_pnp = iOUT_Step)),
             xINtoAS := _20_AUTO.recipe.st120.xUseVerLeft AND
                        (ST120_Feeder_e.rotate_to_feeder = iOUT_Step OR
                        ST120_Feeder_e.Init_pivot_to_feeder = iOUT_Step),
             tIN_ErrAS := DINT_TO_TIME(_20_AUTO.recipe.cylinder2Pos[StationList_e.ST120]
                                           [ST120_Cylinders_e.GreiferLinks].toAS_alarm_time),
             tIN_ErrGS := DINT_TO_TIME(_20_AUTO.recipe.cylinder2Pos[StationList_e.ST120]
                                           [ST120_Cylinders_e.GreiferLinks].toGS_alarm_time),
             tIN_WaitAS := DINT_TO_TIME(_20_AUTO.recipe.cylinder2Pos[StationList_e.ST120]
                                            [ST120_Cylinders_e.GreiferLinks].toAS_wait_time),
             tIN_WaitGS := DINT_TO_TIME(_20_AUTO.recipe.cylinder2Pos[StationList_e.ST120]
                                            [ST120_Cylinders_e.GreiferLinks].toGS_wait_time));

simu_pivotLeft(xIN_Enable := FEEDER_SIMULATION AND CONST.USE_SIMULATION,
               xIN_inGS   := IO_BOX.I6400_ST120_schwenken_links_in_vertikal,
               xIN_inAS   := IO_BOX.I6401_ST120_schwenken_links_in_horizontal,
               xIN_valve  := fb_pivotLeft.xOUT_VALVE,
               tIN_GS_ms  := 500,  //ms
               tIN_AS_ms  := 500); //ms

fb_pivotRight(xIN_Reset    := xIN_Reset OR (ST120_Feeder_e.RESET = iOUT_Step),
              xIN_Quit     := xIN_Quit,
              xIN_Manu     := enState.StateMANU = enIN_State,
              pbtIN_Button := ADR(HMI.btManuCylinders[StationList_e.ST120][4]),
              xIN_GS       := simu_pivotRight.xOUT_inGS,
              xIN_AS       := simu_pivotRight.xOUT_inAS,
              xIN_FREE     := xIN_PnpGripperOpen OR xIN_PnpNotOnTheWay,
              xINtoGS      :=
                  _20_AUTO.recipe.st120.xUseVerRight AND
                  ((ST120_Feeder_e.rotate_to_pnp = iOUT_Step) OR (ST120_Feeder_e.Init_pivot_to_pnp = iOUT_Step)),
              xINtoAS := _20_AUTO.recipe.st120.xUseVerRight AND
                         (ST120_Feeder_e.rotate_to_feeder = iOUT_Step OR
                         ST120_Feeder_e.Init_pivot_to_feeder = iOUT_Step),
              tIN_ErrAS := DINT_TO_TIME(_20_AUTO.recipe.cylinder2Pos[StationList_e.ST120]
                                            [ST120_Cylinders_e.GreiferRechts].toAS_alarm_time),
              tIN_ErrGS := DINT_TO_TIME(_20_AUTO.recipe.cylinder2Pos[StationList_e.ST120]
                                            [ST120_Cylinders_e.GreiferRechts].toGS_alarm_time),
              tIN_WaitAS := DINT_TO_TIME(_20_AUTO.recipe.cylinder2Pos[StationList_e.ST120]
                                             [ST120_Cylinders_e.GreiferRechts].toAS_wait_time),
              tIN_WaitGS := DINT_TO_TIME(_20_AUTO.recipe.cylinder2Pos[StationList_e.ST120]
                                             [ST120_Cylinders_e.GreiferRechts].toGS_wait_time));

simu_pivotRight(xIN_Enable := FEEDER_SIMULATION AND CONST.USE_SIMULATION,
                xIN_inGS   := IO_BOX.I6402_ST120_schwenken_rechts_in_vertikal,
                xIN_inAS   := IO_BOX.I6403_ST120_schwenken_rechts_in_horizontal,
                xIN_valve  := fb_pivotRight.xOUT_VALVE,
                tIN_GS_ms  := 500,  //ms
                tIN_AS_ms  := 500); //ms

btfb_feederLeft(pbtIN  := ADR(HMI.btManuCylinders[StationList_e.ST120][7]),
                xINdis := (enIN_State <> enState.StateMANU),
                xINon  :=,
                xINerr := fb_feederLeft.xOUT_Empty);

IF btfb_feederLeft.pbtIN^.rtrig THEN
    btfb_feederLeft.xINon := NOT btfb_feederLeft.xINon;
ELSIF (enIN_State <> enState.StateMANU) THEN
    btfb_feederLeft.xINon := FALSE;
END_IF;

fb_feederLeft(xIN_Enable := (enIN_State = enState.StateAUTO OR enIN_State = enState.StateSTEP) AND
                            _20_AUTO.recipe.st120.xUseVerLeft,
              // here we do something special. We only want the hublader to run
              // when no piece are at the maxi sensor to prevent a stuck usage 
              xIN_PieceInEnd            := IO_BOX.I8304_ST120_maxi_zufurung_links,
              xIN_PieceMax              := IO_BOX.I8304_ST120_maxi_zufurung_links,
              xIN_InSimulation          := FEEDER_SIMULATION AND CONST.USE_SIMULATION,
              refIN_SimulatedFifo       := simu_fifoLeft,
              iIN_FifoSetMaxSensorValue := BAND_SIZE_FOR_TUBE_LEFT,
              diIN_SignlFilter_ms       := _20_AUTO.recipe.st120.FeederConfigLeft.InFilterDelay,
              diIN_StartDelay_ms        := _20_AUTO.recipe.st120.FeederConfigLeft.StartDelay,
              diIN_StopDelay_ms         := _20_AUTO.recipe.st120.FeederConfigLeft.StopDelay,
              diIN_EmptyDelay_ms        := _20_AUTO.recipe.st120.FeederConfigLeft.EmptyDelay);

btfb_feederRight(pbtIN  := ADR(HMI.btManuCylinders[StationList_e.ST120][8]),
                 xINdis := (enIN_State <> enState.StateMANU),
                 xINon  :=,
                 xINerr := fb_feederRight.xOUT_Empty);

IF btfb_feederRight.pbtIN^.rtrig THEN
    btfb_feederRight.xINon := NOT btfb_feederRight.xINon;
ELSIF (enIN_State <> enState.StateMANU) THEN
    btfb_feederRight.xINon := FALSE;
END_IF;

fb_feederRight(xIN_Enable := (enIN_State = enState.StateAUTO OR enIN_State = enState.StateSTEP) AND
                             _20_AUTO.recipe.st120.xUseVerRight,
               // here we do something special. We only want the hublader to run
               // when no piece are at the maxi sensor to prevent a stuck usage 
               xIN_PieceInEnd            := IO_BOX.I8305_ST120_maxi_zufurung_rechts,
               xIN_PieceMax              := IO_BOX.I8305_ST120_maxi_zufurung_rechts,
               xIN_InSimulation          := FEEDER_SIMULATION AND CONST.USE_SIMULATION,
               refIN_SimulatedFifo       := simu_fifoRight,
               iIN_FifoSetMaxSensorValue := BAND_SIZE_FOR_TUBE_RIGHT,
               diIN_SignlFilter_ms       := _20_AUTO.recipe.st120.FeederConfigRight.InFilterDelay,
               diIN_StartDelay_ms        := _20_AUTO.recipe.st120.FeederConfigRight.StartDelay,
               diIN_StopDelay_ms         := _20_AUTO.recipe.st120.FeederConfigRight.StopDelay,
               diIN_EmptyDelay_ms        := _20_AUTO.recipe.st120.FeederConfigRight.EmptyDelay);

simu_feederLeft(xIN_Enable         := FEEDER_SIMULATION AND CONST.USE_SIMULATION,
                xIN_PceSensor      := IO_BOX.I8304_ST120_maxi_zufurung_links,
                tIN_NewPieceTime   := 500,
                iIN_WaitTimeMin_ms := 1000,
                iIN_WaitTimeMax_ms := 1500);

simu_feederRight(xIN_Enable         := FEEDER_SIMULATION AND CONST.USE_SIMULATION,
                 xIN_PceSensor      := IO_BOX.I8305_ST120_maxi_zufurung_rechts,
                 tIN_NewPieceTime   := 500,
                 iIN_WaitTimeMin_ms := 1000,
                 iIN_WaitTimeMax_ms := 1500);

fb_hubladerLeft(xIN_Reset    := xIN_Reset OR (ST120_Feeder_e.RESET = iOUT_Step),
                xIN_Quit     := xIN_Quit,
                xIN_Manu     := enState.StateMANU = enIN_State,
                pbtIN_Button := ADR(HMI.btManuCylinders[StationList_e.ST120][5]),
                xIN_GS       := simu_hubladerLeft.xOUT_inGS,
                xIN_AS       := simu_hubladerLeft.xOUT_inAS,
                xIN_FREE     := TRUE,
                xINtoGS      := fb_feederLeft.xOUT_EnableFeeder AND fb_hubladerLeft.xIN_AS,
                xINtoAS      := fb_feederLeft.xOUT_EnableFeeder AND fb_hubladerLeft.xIN_GS,
                tIN_ErrAS    := DINT_TO_TIME(_20_AUTO.recipe.cylinder2Pos[StationList_e.ST120]
                                                 [ST120_Cylinders_e.HubladerLinks].toAS_alarm_time),
                tIN_ErrGS := DINT_TO_TIME(_20_AUTO.recipe.cylinder2Pos[StationList_e.ST120]
                                              [ST120_Cylinders_e.HubladerLinks].toGS_alarm_time),
                tIN_WaitAS := DINT_TO_TIME(_20_AUTO.recipe.cylinder2Pos[StationList_e.ST120]
                                               [ST120_Cylinders_e.HubladerLinks].toAS_wait_time),
                tIN_WaitGS := DINT_TO_TIME(_20_AUTO.recipe.cylinder2Pos[StationList_e.ST120]
                                               [ST120_Cylinders_e.HubladerLinks].toGS_wait_time));

simu_hubladerLeft(xIN_Enable := FEEDER_SIMULATION AND CONST.USE_SIMULATION,
                  xIN_inGS   := IO_BOX.I8204_ST120_hublader_links_unten,
                  xIN_inAS   := IO_BOX.I8205_ST120_hublader_links_oben,
                  xIN_valve  := fb_hubladerLeft.xOUT_VALVE,
                  tIN_GS_ms  := 800,  //ms
                  tIN_AS_ms  := 800); //ms

fb_hubladerRight(xIN_Reset    := xIN_Reset OR (ST120_Feeder_e.RESET = iOUT_Step),
                 xIN_Quit     := xIN_Quit,
                 xIN_Manu     := enState.StateMANU = enIN_State,
                 pbtIN_Button := ADR(HMI.btManuCylinders[StationList_e.ST120][6]),
                 xIN_GS       := simu_hubladerRight.xOUT_inGS,
                 xIN_AS       := simu_hubladerRight.xOUT_inAS,
                 xIN_FREE     := TRUE,
                 xINtoGS      := fb_feederRight.xOUT_EnableFeeder AND fb_hubladerRight.xIN_AS,
                 xINtoAS      := fb_feederRight.xOUT_EnableFeeder AND fb_hubladerRight.xIN_GS,
                 tIN_ErrAS    := DINT_TO_TIME(_20_AUTO.recipe.cylinder2Pos[StationList_e.ST120]
                                                  [ST120_Cylinders_e.HubladerRechts].toAS_alarm_time),
                 tIN_ErrGS := DINT_TO_TIME(_20_AUTO.recipe.cylinder2Pos[StationList_e.ST120]
                                               [ST120_Cylinders_e.HubladerRechts].toGS_alarm_time),
                 tIN_WaitAS := DINT_TO_TIME(_20_AUTO.recipe.cylinder2Pos[StationList_e.ST120]
                                                [ST120_Cylinders_e.HubladerRechts].toAS_wait_time),
                 tIN_WaitGS := DINT_TO_TIME(_20_AUTO.recipe.cylinder2Pos[StationList_e.ST120]
                                                [ST120_Cylinders_e.HubladerRechts].toGS_wait_time));

simu_hubladerRight(xIN_Enable := FEEDER_SIMULATION AND CONST.USE_SIMULATION,
                   xIN_inGS   := IO_BOX.I8300_ST120_hublader_rechts_unten,
                   xIN_inAS   := IO_BOX.I8301_ST120_hublader_rechts_oben,
                   xIN_valve  := fb_hubladerRight.xOUT_VALVE,
                   tIN_GS_ms  := 800,  //ms
                   tIN_AS_ms  := 800); //ms

rtPutPieceLeft(CLK := simu_hubladerLeft.xOUT_inAS);
rtPutPieceRight(CLK := simu_hubladerRight.xOUT_inAS);

IF rtPutPieceLeft.Q THEN
    simu_fifoLeft.Put(1);
END_IF

IF rtPutPieceRight.Q THEN
    simu_fifoRight.Put(1);
END_IF

(*******************************************************************)
(* OUTPUTS *)
(*******************************************************************)
// Error Flag 
xOUT_ErrFlag := (bOUT_Error <> 0) OR (ST120_Feeder_e.ERROR = iOUT_Step);
// Baustein befindet sich im Ablauf 
xOUT_Busy := (iOUT_Step > ST120_Feeder_e.READY) AND (iOUT_Step < ST120_Feeder_e.DONE);
// Baustein hat den Ablauf beendet
xOUT_Done := (iOUT_Step = ST120_Feeder_e.DONE);
// Process ready
xOUT_Ready := (iOUT_Step = ST120_Feeder_e.READY);
// Timeout FB 				 		
xOUT_Timeout := TON_Timeout.Q;
// Itialisierung fertig			
xOUT_InitDone := (iOUT_Step = ST120_Feeder_e.READY);
// Aktueller Schritt			
iOUT_Step := iOUT_Step; //Im Ablauf gesetzt		
sOUT_Step := TO_STRING(iOUT_Step);
//Fehlernummer	 
bOUT_Error := bOUT_Error; //Im Ablauf/FB gesetzt	
(* Warte (alle Schritte wo auf FG oder Teile gewartet wird) *)
xOUT_Wait := (iOUT_Step = ST120_Feeder_e.DONE) OR
             (iOUT_Step = ST120_Feeder_e.READY);

IO_BOX.Q5204_14_ST120_schwenken_links :=
    fb_pivotLeft.xOUT_VALVE AND NOT (FEEDER_SIMULATION AND CONST.USE_SIMULATION);

IO_BOX.Q5205_14_ST120_schwenken_rechts :=
    fb_pivotRight.xOUT_VALVE AND NOT (FEEDER_SIMULATION AND CONST.USE_SIMULATION);

IO_BOX.Q8207_ST120_hublader_links_valve :=
    fb_hubladerLeft.xOUT_VALVE AND NOT (FEEDER_SIMULATION AND CONST.USE_SIMULATION);

IO_BOX.Q8303_ST120_hublader_rechts_valve :=
    fb_hubladerRight.xOUT_VALVE AND NOT (FEEDER_SIMULATION AND CONST.USE_SIMULATION);

IO_BOX.Q8201_ST120_forderband_ein_l :=
    (enIN_State >= enState.StateLEER) AND
    pxFG_Freigabe^ AND
    NOT (FEEDER_SIMULATION AND CONST.USE_SIMULATION);

IO_BOX.Q8203_ST120_forderband_ein_r :=
    (enIN_State >= enState.StateLEER) AND
    pxFG_Freigabe^ AND
    NOT (FEEDER_SIMULATION AND CONST.USE_SIMULATION);

(*******************************************************************)
(* Ablauf *)
(*******************************************************************)

(* Sperren *)
IF xIN_Sperre THEN
    iPreStep  := ST120_Feeder_e.RESET;
    iOUT_Step := ST120_Feeder_e.RESET;
    RETURN;
END_IF;

(* Schritt Merker *)
IF iAktStep <> iOUT_Step THEN
    iLastStep := iAktStep;
    iAktStep  := iOUT_Step;
END_IF

(* START *)
rtSTART(CLK := xIN_Start);

(* error management *)
IF 0 = bOUT_Error THEN
    IF fb_pivotLeft.xOUT_ErrFlag THEN
        bOUT_Error := ST120_Alarm_e.Cylinder_pivot_left;
    ELSIF fb_pivotRight.xOUT_ErrFlag THEN
        bOUT_Error := ST120_Alarm_e.Cylinder_pivot_right;
    ELSIF fb_hubladerLeft.xOUT_ErrFlag THEN
        bOUT_Error := ST120_Alarm_e.Cylinder_hublader_left;
    ELSIF fb_hubladerRight.xOUT_ErrFlag THEN
        bOUT_Error := ST120_Alarm_e.Cylinder_hublader_right;
    END_IF
ELSIF iOUT_Step < ST120_Feeder_e.ERROR THEN
    iOUT_Step := ST120_Feeder_e.ERROR;
END_IF

(*******************************************************************)
(* Schrittkette  *)
(*******************************************************************)
CASE iOUT_Step OF

(***** RESET *****)
ST120_Feeder_e.RESET: (* Schritt 0-99 *)
    //Initialisierungen
    //Start Init Ablauf
    IF xIN_Init THEN
        iOUT_Step := ST120_Feeder_e.INIT;
        //Start Manu Ablauf
    ELSIF enIN_State = StateMANU AND xIN_NextStep THEN
        iOUT_Step := ST120_Feeder_e.INIT;
    END_IF;

(***** INIT *****)
ST120_Feeder_e.INIT: (* Grundstellung ? *)
    IF xIN_PnpGripperOpen AND xIN_PnpNotOnTheWay THEN
        iOUT_Step := ST120_Feeder_e.Init_pneumatics;
    END_IF;

ST120_Feeder_e.Init_pneumatics:
    // TODO check all the sensors
    IF FEEDER_SIMULATION AND CONST.USE_SIMULATION THEN
        iOUT_Step := ST120_Feeder_e.Init_pivot_to_feeder;
    ELSE
        IF (NOT _20_AUTO.recipe.st120.xUseVerLeft AND IO_BOX.I6404_ST120_teil_in_vereizelung_links) OR
           (NOT _20_AUTO.recipe.st120.xUseVerRight AND IO_BOX.I6405_ST120_teil_in_vereinzelung_rechts) THEN
            bOUT_Error := ST120_Alarm_e.Piece_in_unused_pivot;
            iOUT_Step  := ST120_Feeder_e.ERROR;

        ELSIF (IO_BOX.I6401_ST120_schwenken_links_in_horizontal AND
               IO_BOX.I6403_ST120_schwenken_rechts_in_horizontal) THEN
            iOUT_Step := ST120_Feeder_e.Init_pivot_to_feeder;

        ELSIF (_20_AUTO.recipe.st120.xUseVerLeft AND NOT IO_BOX.I6404_ST120_teil_in_vereizelung_links) AND
              (_20_AUTO.recipe.st120.xUseVerRight AND IO_BOX.I6405_ST120_teil_in_vereinzelung_rechts) THEN
            bOUT_Error := ST120_Alarm_e.Piece_missing_left_pivot;
            iOUT_Step  := ST120_Feeder_e.ERROR;

        ELSIF (_20_AUTO.recipe.st120.xUseVerLeft AND IO_BOX.I6404_ST120_teil_in_vereizelung_links) AND
              (_20_AUTO.recipe.st120.xUseVerRight AND NOT IO_BOX.I6405_ST120_teil_in_vereinzelung_rechts) THEN
            bOUT_Error := ST120_Alarm_e.Piece_missing_right_pivor;
            iOUT_Step  := ST120_Feeder_e.ERROR;

        ELSIF NOT IO_BOX.I6404_ST120_teil_in_vereizelung_links AND NOT IO_BOX.I6405_ST120_teil_in_vereinzelung_rechts
            THEN
            iOUT_Step := ST120_Feeder_e.Init_pivot_to_feeder;

        ELSE
            iOUT_Step := ST120_Feeder_e.Init_pivot_to_pnp;
        END_IF
    END_IF

ST120_Feeder_e.Init_pivot_to_feeder:
    IF (NOT _20_AUTO.recipe.st120.xUseVerLeft OR fb_pivotLeft.xOUT_inAS) AND
       (NOT _20_AUTO.recipe.st120.xUseVerRight OR fb_pivotRight.xOUT_inAS) THEN
        iOUT_Step := ST120_Feeder_e.READY;
    END_IF

ST120_Feeder_e.Init_pivot_to_pnp:
    IF (NOT _20_AUTO.recipe.st120.xUseVerLeft OR fb_pivotLeft.xOUT_inGS) AND
       (NOT _20_AUTO.recipe.st120.xUseVerRight OR fb_pivotRight.xOUT_inGS) THEN
        iOUT_Step := ST120_Feeder_e.READY;
    END_IF

(***** READY / INIT DONE *****)
ST120_Feeder_e.READY: (* Start AUTO,END,LEER,STEP *)
    IF xIN_Start THEN //IF rtSTART.Q THEN
        iOUT_Step := ST120_Feeder_e.START;
    END_IF

(***** START  ZYKLISCH *****)
ST120_Feeder_e.START: (*  *)
    IF xIN_NextStep AND pxFG_Freigabe^ THEN
        iOUT_Step := ST120_Feeder_e.wait_tube_presence;
    END_IF;

ST120_Feeder_e.wait_tube_presence:
    IF (FEEDER_SIMULATION AND CONST.USE_SIMULATION) THEN
        IF (NOT _20_AUTO.recipe.st120.xUseVerLeft OR (simu_fifoLeft.GetLen() >= BAND_SIZE_FOR_TUBE_LEFT)) AND
           (NOT _20_AUTO.recipe.st120.xUseVerRight OR (simu_fifoRight.GetLen() >= BAND_SIZE_FOR_TUBE_RIGHT)) THEN
            iOUT_Step := ST120_Feeder_e.wait_pnp_ready;
        END_IF

    ELSE
        IF (NOT _20_AUTO.recipe.st120.xUseVerLeft OR TON_PieceInPivotLeft.Q) AND
           (NOT _20_AUTO.recipe.st120.xUseVerRight OR TON_PieceInPivotRight.Q) THEN
            iOUT_Step := ST120_Feeder_e.wait_pnp_ready;
        END_IF
    END_IF

ST120_Feeder_e.wait_pnp_ready:
    IF xIN_PnpGripperOpen THEN
        iOUT_Step := ST120_Feeder_e.rotate_to_pnp;
    END_IF

ST120_Feeder_e.rotate_to_pnp:
    IF fb_pivotLeft.xOUT_inGS AND fb_pivotRight.xOUT_inGS THEN
        iOUT_Step := ST120_Feeder_e.wait_pce_picked;
    END_IF

ST120_Feeder_e.wait_pce_picked:
    IF xIN_PickPiece THEN
        IF _20_AUTO.recipe.st120.xUseVerLeft THEN
            simu_fifoLeft.Pop(1);
        END_IF

        IF _20_AUTO.recipe.st120.xUseVerRight THEN
            simu_fifoRight.Pop(1);
        END_IF

        iOUT_Step := ST120_Feeder_e.wait_pnp_move_out_with_the_piece;
    END_IF

ST120_Feeder_e.wait_pnp_move_out_with_the_piece:
    IF xIN_PnpNotOnTheWay THEN
        iOUT_Step := ST120_Feeder_e.rotate_to_feeder;
    END_IF

ST120_Feeder_e.rotate_to_feeder:
    IF (NOT _20_AUTO.recipe.st120.xUseVerLeft OR fb_pivotLeft.xOUT_inAS) AND
       (NOT _20_AUTO.recipe.st120.xUseVerRight OR fb_pivotRight.xOUT_inAS) THEN
        iOUT_Step := ST120_Feeder_e.DONE;
    END_IF

(***** DONE *****)
ST120_Feeder_e.DONE: (* Letzter Schritt  *)
    IF NOT xIN_AlarmAktiv THEN
        //AUTO
        IF (enIN_State = StateAUTO) AND xIN_RestartCYCL THEN
            iOUT_Step := ST120_Feeder_e.START;
            //STEP / END / LEERFAHREN restart
        ELSIF (enIN_State < StateAUTO) AND (enIN_State >= enState.StateSTEP) AND xIN_RestartCYCL THEN
            iOUT_Step := ST120_Feeder_e.START;
            //STEP / END / LEERFAHREN fertig
        ELSIF (enIN_State = StateREADY) THEN
            iOUT_Step := ST120_Feeder_e.READY;
        END_IF;
    END_IF;

(************ ERROR *************)
ST120_Feeder_e.ERROR: (* ERROR *) ;

END_CASE;

END_FUNCTION_BLOCK

// ---- POUs/20_AUTO/ST120/FB_ABL_120_Pnp.TcPOU
FUNCTION_BLOCK FB_ABL_120_Pnp
(****************************************************************************************)
(*	TITEL				laden kristall- Modul	    										*)
(*	Status				ungetestet                         								*)
(*	Beschrieb:			Ablaufbeschreibung												*)
(*																						*)
(*	Steps:	self-explained using enum													*)
(***********************************Revisionen*******************************************)
(*	see github blames																	*)
(****************************************************************************************)

VAR_INPUT
    xIN_Reset       : BOOL;          // Schrittkette zurücksetzen 
    xIN_Init        : BOOL;          // Initialisieren
    xIN_Quit        : BOOL;          // Fehler quittieren 
    xIN_Start       : BOOL;          // Startbefehl
    xIN_Sperre      : BOOL;          // FB Sperren 
    xIN_NextStep    : BOOL;          // Nächsten Schritt ausführen 
    xIN_AlarmAktiv  : BOOL;          // Anlage hat Alarm
    xIN_DryCycle    : BOOL;          // Fahren ohne Teile
    xIN_RestartCYCL : BOOL;          // Zyklus erneut starten im STEP, END, LEERFAHREN
    enIN_State      : enState;       // Status Anlage
    tIN_Timeout     : TIME := T#10s; // Timout

    pxFG_Freigabe : POINTER TO BOOL; //Freigabe von Station

    // Application specific
    Mover              : REFERENCE TO FB_Mover;
    xIN_PceReadyToPick : BOOL; // the piece(s) is/are ready to picked
END_VAR
VAR_OUTPUT
    (* standart Ausgänge *)
    xOUT_ErrFlag  : BOOL;        // Error Flag 
    xOUT_Busy     : BOOL;        // Baustein befindet sich im Ablauf 
    xOUT_Done     : BOOL;        // Baustein hat den Ablauf beendet 		
    xOUT_Ready    : BOOL;        // Ready to begin, should be the same state as done	
    xOUT_Timeout  : BOOL;        // Timeout FB 
    xOUT_InitDone : BOOL;        // initialisierung fertig
    xOUT_Wait     : BOOL;        // Wartet auf Bedingung
    iOUT_Step     : ST120_Pnp_e; // Aktueller Schritt 
    sOUT_Step     : STRING;      // Aktueller Schritt but in string format
    bOUT_Error    : BYTE;        // Fehlernummer

    iOUT_ProcessCompletion : INT;  //process completion, express in % (0-100)
    xOUT_MoverFree         : BOOL; // The mover is free to move
    xOUT_PickPiece         : BOOL; // Set to true when a piece is picked

END_VAR
VAR
    (* Standard *)
    (* Schritt *)
    iLastStep : ST120_Pnp_e; // Merker letzter Schritt 
    iPreStep  : ST120_Pnp_e; // Schritt zurück nach Alarm 
    iAktStep  : ST120_Pnp_e; // aktueller Schritt

    // Trigger Starten 
    rtSTART : R_TRIG;
    // Timer TimeOut 
    TON_Timeout : TON;

    (* Bausteine *)

    (* Spezial *)
    fb_axis120_01Y : FB_AxisLM_V1_1;
    fb_axis120_02Z : FB_AxisLM_V1_1;

    fb_PnpHorAxis : FB_LinearMotionMan;
    fb_PnpVerAxis : FB_LinearMotionMan;

    fb_gripperLeft    : FB_ZylMo2El_V2_1;
    fb_gripperRight   : FB_ZylMo2El_V2_1;
    simu_gripperLeft  : FB_Simu_Zyl2Pos;
    simu_gripperRight : FB_Simu_Zyl2Pos;

    fb_simu_axis120_01Y : FB_Simu_AxisLM_V1_1;
    fb_simu_axis120_02Z : FB_Simu_AxisLM_V1_1;

END_VAR
VAR CONSTANT
    PNP_SIMULATION : BOOL := FALSE; // Set to TRUE to simulate this part of the program
END_VAR

(*******************************************************************)
(* Trigger  *)
(*******************************************************************)
(* Zurücksetzen *)
IF xIN_RESET THEN
    iPreStep  := ST120_Pnp_e.RESET;
    iOUT_Step := ST120_Pnp_e.RESET;
END_IF

(* Error Quittieren *)
IF (bOUT_Error <> 0) AND xIN_Quit THEN
    xOUT_ErrFlag := FALSE;
    bOUT_Error   := 0;
    iOUT_Step    := iPreStep;
END_IF

(*******************************************************************)
(* Timer *)
(*******************************************************************)
TON_Timeout(IN := xIN_NextStep AND (iLastStep = iOUT_Step) (*todo FG *) ,
            PT := tIN_Timeout);

(*******************************************************************)
(* Bausteine *)
(*******************************************************************)
fb_PnpHorAxis(config          := _20_AUTO.recipe.linearAxis[LinearAxis_e.ST120_01Y],
              xIN_Init        := enIN_State = enState.StateINIT,
              xIN_Reset       := xIN_Reset,
              lrIN_CurrPos    := fb_axis120_01Y.rOUT_ActPos,
              lrIN_Delta_mm   := 0.5,
              iIN_CurrentStep := iOUT_Step,
              iIN_moveNumber  := ST120_PnpHorPos_e._max);

fb_simu_axis120_01Y(xIN_Enable          := PNP_SIMULATION AND CONST.USE_SIMULATION,
                    bIN_AxisCntr        := fb_axis120_01Y.bOUT_AxisCntr,
                    wIN_AxisState       := ST120_Axis.axis120_01Y.wState,
                    udiIN_HomingTime_ms := 2000,
                    pIN_axisSimu        := ADR(SIMU.axis_ref[Axis_e.ST120_01Y]),
                    pIN_axisHW          := ADR(ST120_Axis.axis120_01Y.axis),
                    rIN_PosActual       := fb_axis120_01Y.rOUT_ActPos,
                    rIN_PosMax          := ST120_Axis.const120_01Y.POS_MAX,
                    rIN_PosMin          := ST120_Axis.const120_01Y.POS_MIN,
                    rIN_PixMax          := 100,
                    rIN_PixMin          := 0);

fb_axis120_01Y(enIN_State       := enIN_State,
               parIN_Buttons    := ADR(AXIS.btTeachArAxis[Axis_e.ST120_01Y]),
               xIN_DisButtons   :=,
               xIN_Quit         := xIN_Quit,
               xIN_PARAMok      := TRUE, (*TODO*)
               xIN_FREE         := TRUE,
               xIN_FREE_HOME    := TRUE,
               rIN_POSMIN       := ST120_Axis.const120_01Y.POS_MIN,
               rIN_POSMAX       := ST120_Axis.const120_01Y.POS_MAX,
               rIN_VELOMAX      := ST120_Axis.const120_01Y.VELO_MAX,
               rIN_VELOMANU     := ST120_Axis.const120_01Y.VELO_MANU,
               rIN_VELOOPEN     := ST120_Axis.const120_01Y.VELO_MANU / 4,
               rIN_JogInc       := AXIS.rTeachIncAxis,
               xIN_Execute      := fb_PnpHorAxis.xOUT_Execute,
               xIN_Home         := ST120_Pnp_e.Init_HomeHorizontals = iAktStep,
               xIN_Relative     :=,
               rIN_Position     := TO_REAL(fb_PnpHorAxis.OUT_MoveProfile.lrPosition),
               rIN_Velocity     := TO_REAL(fb_PnpHorAxis.OUT_MoveProfile.lrVelocity),
               rIN_Acceleration := TO_REAL(fb_PnpHorAxis.OUT_MoveProfile.lrAccel),
               rIN_Deceleration := TO_REAL(fb_PnpHorAxis.OUT_MoveProfile.lrDecel),
               rIN_Jerk         := TO_REAL(fb_PnpHorAxis.OUT_MoveProfile.lrJerk),
               rIN_PosManu      :=
               TO_REAL(_20_AUTO.recipe
                           .linearAxis[LinearAxis_e.ST120_01Y].movesList[AXIS.bTeachPos[Axis_e.ST120_01Y]].lrPosition),
               rIN_VeloJogManu := TO_REAL(Axis.rJogVelo_pc),
               xIN_Reset       := (ST120_Pnp_e.RESET = iAktStep) OR xIN_Reset,
               // the simu fb gives the hardware signal when the simulation is disabled
               wAxisState    := fb_simu_axis120_01Y.wOUT_AxisState,
               bOUT_AxisCntr => ST120_Axis.axis120_01Y.bCtrlHi,
               rOUT_ActPos   => ST120_Axis.axis120_01Y.rActPos,
               axisIN_REF    := fb_simu_axis120_01Y.pOUT_axisRef^);

fb_PnpVerAxis(config          := _20_AUTO.recipe.linearAxis[LinearAxis_e.ST120_02Z],
              xIN_Init        := enIN_State = enState.StateINIT,
              xIN_Reset       := xIN_Reset,
              lrIN_CurrPos    := fb_axis120_02Z.rOUT_ActPos,
              lrIN_Delta_mm   := 0.5,
              iIN_CurrentStep := iOUT_Step,
              iIN_moveNumber  := ST120_PnpVerPos_e._max);

fb_simu_axis120_02Z(xIN_Enable          := PNP_SIMULATION AND CONST.USE_SIMULATION,
                    bIN_AxisCntr        := fb_axis120_02Z.bOUT_AxisCntr,
                    wIN_AxisState       := ST120_Axis.axis120_02Z.wState,
                    udiIN_HomingTime_ms := 2000,
                    pIN_axisSimu        := ADR(SIMU.axis_ref[Axis_e.ST120_02Z]),
                    pIN_axisHW          := ADR(ST120_Axis.axis120_02Z.axis),
                    rIN_PosActual       := fb_axis120_02Z.rOUT_ActPos,
                    rIN_PosMax          := ST120_Axis.const120_02Z.POS_MAX,
                    rIN_PosMin          := ST120_Axis.const120_02Z.POS_MIN,
                    rIN_PixMax          := 100,
                    rIN_PixMin          := 0);

fb_axis120_02Z(enIN_State       := enIN_State,
               parIN_Buttons    := ADR(AXIS.btTeachArAxis[Axis_e.ST120_02Z]),
               xIN_DisButtons   :=,
               xIN_Quit         := xIN_Quit,
               xIN_PARAMok      := TRUE, (*TODO*)
               xIN_FREE         := TRUE,
               xIN_FREE_HOME    := TRUE,
               rIN_POSMIN       := ST120_Axis.const120_02Z.POS_MIN,
               rIN_POSMAX       := ST120_Axis.const120_02Z.POS_MAX,
               rIN_VELOMAX      := ST120_Axis.const120_02Z.VELO_MAX,
               rIN_VELOMANU     := ST120_Axis.const120_02Z.VELO_MANU,
               rIN_VELOOPEN     := ST120_Axis.const120_02Z.VELO_MANU / 4,
               rIN_JogInc       := AXIS.rTeachIncAxis,
               xIN_Execute      := fb_PnpVerAxis.xOUT_Execute,
               xIN_Home         := ST120_Pnp_e.Init_HomeVerticals = iAktStep,
               xIN_Relative     :=,
               rIN_Position     := TO_REAL(fb_PnpVerAxis.OUT_MoveProfile.lrPosition),
               rIN_Velocity     := TO_REAL(fb_PnpVerAxis.OUT_MoveProfile.lrVelocity),
               rIN_Acceleration := TO_REAL(fb_PnpVerAxis.OUT_MoveProfile.lrAccel),
               rIN_Deceleration := TO_REAL(fb_PnpVerAxis.OUT_MoveProfile.lrDecel),
               rIN_Jerk         := TO_REAL(fb_PnpVerAxis.OUT_MoveProfile.lrJerk),
               rIN_PosManu      :=
               TO_REAL(_20_AUTO.recipe
                           .linearAxis[LinearAxis_e.ST120_02Z].movesList[AXIS.bTeachPos[Axis_e.ST120_02Z]].lrPosition),
               rIN_VeloJogManu := TO_REAL(Axis.rJogVelo_pc),
               xIN_Reset       := (ST120_Pnp_e.RESET = iAktStep) OR xIN_Reset,
               // the simu fb gives the hardware signal when the simulation is disabled
               wAxisState    := fb_simu_axis120_02Z.wOUT_AxisState,
               bOUT_AxisCntr => ST120_Axis.axis120_02Z.bCtrlHi,
               rOUT_ActPos   => ST120_Axis.axis120_02Z.rActPos,
               axisIN_REF    := fb_simu_axis120_02Z.pOUT_axisRef^);

fb_gripperLeft(xIN_Reset    := xIN_Reset OR (ST120_Pnp_e.RESET = iOUT_Step),
               xIN_Quit     := xIN_Quit,
               xIN_Manu     := enState.StateMANU = enIN_State,
               pbtIN_Button := ADR(HMI.btManuCylinders[StationList_e.ST120][1]),
               xIN_GS       := simu_gripperLeft.xOUT_inGS,
               xIN_AS       := simu_gripperLeft.xOUT_inAS,
               xIN_FREE     := TRUE,
               xINtoGS      := _20_AUTO.recipe.st120.xUseVerLeft AND ST120_Pnp_e.Gripper_close = iOUT_Step,
               xINtoAS      := (ST120_Pnp_e.Gripper_open = iOUT_Step) OR
                               (ST120_Pnp_e.Init_open_left_clamp = iOUT_Step),
               tIN_ErrAS := DINT_TO_TIME(_20_AUTO.recipe.cylinder2Pos[StationList_e.ST120]
                                             [ST120_Cylinders_e.GreiferLinks].toAS_alarm_time),
               tIN_ErrGS := DINT_TO_TIME(_20_AUTO.recipe.cylinder2Pos[StationList_e.ST120]
                                             [ST120_Cylinders_e.GreiferLinks].toGS_alarm_time),
               tIN_WaitAS := DINT_TO_TIME(_20_AUTO.recipe.cylinder2Pos[StationList_e.ST120]
                                              [ST120_Cylinders_e.GreiferLinks].toAS_wait_time),
               tIN_WaitGS := DINT_TO_TIME(_20_AUTO.recipe.cylinder2Pos[StationList_e.ST120]
                                              [ST120_Cylinders_e.GreiferLinks].toGS_wait_time));

simu_gripperLeft(xIN_Enable := TRUE, // PNP_SIMULATION AND CONST.USE_SIMULATION,
                 xIN_inGS   := IO_BOX.I6300_ST120_greifer_links_geschlossen,
                 xIN_inAS   := IO_BOX.I6301_ST120_greifer_links_offen,
                 xIN_valve  := fb_gripperLeft.xOUT_VALVE,
                 tIN_GS_ms  := 200,  //ms
                 tIN_AS_ms  := 200); //ms

fb_gripperRight(xIN_Reset    := xIN_Reset OR (ST120_Pnp_e.RESET = iOUT_Step),
                xIN_Quit     := xIN_Quit,
                xIN_Manu     := enState.StateMANU = enIN_State,
                pbtIN_Button := ADR(HMI.btManuCylinders[StationList_e.ST120][2]),
                xIN_GS       := simu_gripperRight.xOUT_inGS,
                xIN_AS       := simu_gripperRight.xOUT_inAS,
                xIN_FREE     := TRUE,
                xINtoGS      := _20_AUTO.recipe.st120.xUseVerRight AND (ST120_Pnp_e.Gripper_close = iOUT_Step),
                xINtoAS      := (ST120_Pnp_e.Gripper_open = iOUT_Step) OR
                                (ST120_Pnp_e.Init_open_right_clamp = iOUT_Step),
                tIN_ErrAS := DINT_TO_TIME(_20_AUTO.recipe.cylinder2Pos[StationList_e.ST120]
                                              [ST120_Cylinders_e.GreiferRechts].toAS_alarm_time),
                tIN_ErrGS := DINT_TO_TIME(_20_AUTO.recipe.cylinder2Pos[StationList_e.ST120]
                                              [ST120_Cylinders_e.GreiferRechts].toGS_alarm_time),
                tIN_WaitAS := DINT_TO_TIME(_20_AUTO.recipe.cylinder2Pos[StationList_e.ST120]
                                               [ST120_Cylinders_e.GreiferRechts].toAS_wait_time),
                tIN_WaitGS := DINT_TO_TIME(_20_AUTO.recipe.cylinder2Pos[StationList_e.ST120]
                                               [ST120_Cylinders_e.GreiferRechts].toGS_wait_time));

simu_gripperRight(xIN_Enable := TRUE, // PNP_SIMULATION AND CONST.USE_SIMULATION,
                  xIN_inGS   := IO_BOX.I6302_ST120_greifer_rechts_geschlossen,
                  xIN_inAS   := IO_BOX.I6303_ST120_greifer_rechts_offen,
                  xIN_valve  := fb_gripperRight.xOUT_VALVE,
                  tIN_GS_ms  := 200,  //ms
                  tIN_AS_ms  := 200); //ms

(*******************************************************************)
(* OUTPUTS *)
(*******************************************************************)
// Error Flag 
xOUT_ErrFlag := (bOUT_Error <> 0) OR (ST120_Pnp_e.ERROR = iOUT_Step);
// Baustein befindet sich im Ablauf 
xOUT_Busy := (iOUT_Step > ST120_Pnp_e.READY) AND (iOUT_Step < ST120_Pnp_e.DONE);
// Baustein hat den Ablauf beendet
xOUT_Done := (iOUT_Step = ST120_Pnp_e.DONE);
// Process ready
xOUT_Ready := (iOUT_Step = ST120_Pnp_e.READY) OR (iOUT_Step = ST120_Pnp_e.waitOnMover);
// Timeout FB 				 		
xOUT_Timeout := TON_Timeout.Q;
// Itialisierung fertig			
xOUT_InitDone := (iOUT_Step = ST120_Pnp_e.READY) OR (iOUT_Step = ST120_Pnp_e.waitOnMover);
// Aktueller Schritt			
iOUT_Step := iOUT_Step; //Im Ablauf gesetzt		
sOUT_Step := TO_STRING(iOUT_Step);
//Fehlernummer	 
bOUT_Error := bOUT_Error; //Im Ablauf/FB gesetzt	
(* Warte (alle Schritte wo auf FG oder Teile gewartet wird) *)
xOUT_Wait := (iOUT_Step = ST120_Pnp_e.DONE) OR
             (iOUT_Step = ST120_Pnp_e.READY) OR
             (iOUT_Step = ST120_Pnp_e.START) OR
             (iOUT_Step = ST120_Pnp_e.waitOnMover) OR
             (iOUT_Step = ST120_Pnp_e.SYNC_MOVER_LEAVE) OR
             (iOUT_Step = ST120_Pnp_e.PnP_WaitOnFeeder);

xOUT_MoverFree := iOUT_Step >= ST120_Pnp_e.MOVER_FREE_OP AND iOUT_Step < ST120_Pnp_e.MOVER_NEEDED_OP;

iOUT_ProcessCompletion := F_GetPercent_2(iAktStep,
                                         ST120_Pnp_e.PnP_Hor_ToRotTablePos,
                                         ST120_Pnp_e.PnP_Hor_ToTrackPos,
                                         ST120_Pnp_e.PnP_Ver_ShuttleDown,
                                         ST120_Pnp_e.PnP_Ver_ShuttleUp);

xOUT_PickPiece := iOUT_Step = ST120_Pnp_e.PnP_Ver_RotTableUp;

IO_BOX.Q5202_14_ST120_greifer_links  := fb_gripperLeft.xOUT_VALVE AND NOT (PNP_SIMULATION AND CONST.USE_SIMULATION);
IO_BOX.Q5203_14_ST120_greifer_rechts := fb_gripperRight.xOUT_VALVE AND NOT (PNP_SIMULATION AND CONST.USE_SIMULATION);

IO_BOX.Q5212_14_ST120_stop_vertical_axis := NOT fb_simu_axis120_02Z.pIN_axisHW^.Status.Error AND
                                            _02_SAFETY.xOUT_ESout AND
                                            _02_SAFETY.xOUT_MonOut AND
                                            NOT (PNP_SIMULATION AND CONST.USE_SIMULATION);

(*******************************************************************)
(* Ablauf *)
(*******************************************************************)

(* Sperren *)
IF xIN_Sperre THEN
    iPreStep  := ST120_Pnp_e.RESET;
    iOUT_Step := ST120_Pnp_e.RESET;
    RETURN;
END_IF;

(* Schritt Merker *)
IF iAktStep <> iOUT_Step THEN
    iLastStep := iAktStep;
    iAktStep  := iOUT_Step;
END_IF

(* START *)
rtSTART(CLK := xIN_Start);

IF 0 = bOUT_Error THEN
    IF fb_axis120_01Y.xOUT_ErrFlag THEN
        bOUT_Error := ST120_Alarm_e.Axis_120_01Y_error;
    ELSIF fb_axis120_02Z.xOUT_ErrFlag THEN
        bOUT_Error := ST120_Alarm_e.Axis_120_02Z_error;
    ELSIF fb_gripperLeft.xOUT_ErrFlag THEN
        bOUT_Error := ST120_Alarm_e.Cylinder_griper_left;
    ELSIF fb_gripperRight.xOUT_ErrFlag THEN
        bOUT_Error := ST120_Alarm_e.Cylinder_griper_right;
    END_IF
ELSIF iOUT_Step < ST120_Pnp_e.ERROR THEN
    iOUT_Step := ST120_Pnp_e.ERROR;
END_IF

(*******************************************************************)
(* Schrittkette  *)
(*******************************************************************)
CASE iOUT_Step OF

(***** RESET *****)
ST120_Pnp_e.RESET: (* Schritt 0-99 *)
    //Initialisierungen
    //Start Init Ablauf
    IF xIN_Init THEN
        iOUT_Step := ST120_Pnp_e.INIT;
        //Start Manu Ablauf
    ELSIF enIN_State = StateMANU AND xIN_NextStep THEN
        iOUT_Step := ST120_Pnp_e.INIT;
    END_IF;

(***** INIT *****)
ST120_Pnp_e.INIT: (* Grundstellung ? *)
    IF fb_axis120_02Z.xOUT_HOMED THEN
        iOUT_Step := ST120_Pnp_e.Init_VerticalsUp;
    ELSE
        iOUT_Step := ST120_Pnp_e.Init_HomeVerticals;
    END_IF

ST120_Pnp_e.Init_HomeVerticals:
    IF fb_axis120_02Z.xOUT_HOMED THEN
        iOUT_Step := ST120_Pnp_e.Init_VerticalsUp;
    END_IF

ST120_Pnp_e.Init_VerticalsUp:
    IF fb_gripperLeft.xIN_AS OR fb_gripperRight.xIN_AS THEN
        IF fb_PnpVerAxis.MoveTo(ST120_PnpVerPos_e.UpFull).xOUT_InPos THEN
            IF fb_axis120_01Y.xOUT_READY OR fb_axis120_01Y.xOUT_HOMED THEN
                iOUT_Step := ST120_Pnp_e.Init_HorizontalsToTrack;
            ELSE
                iOUT_Step := ST120_Pnp_e.Init_HomeHorizontals;
            END_IF
        END_IF
    ELSE
        IF fb_PnpVerAxis.MoveTo(ST120_PnpVerPos_e.UpEmpty).xOUT_InPos THEN
            IF fb_axis120_01Y.xOUT_READY OR fb_axis120_01Y.xOUT_HOMED THEN
                iOUT_Step := ST120_Pnp_e.Init_HorizontalsToTrack;
            ELSE
                iOUT_Step := ST120_Pnp_e.Init_HomeHorizontals;
            END_IF
        END_IF
    END_IF

ST120_Pnp_e.Init_HomeHorizontals:
    IF fb_axis120_01Y.xOUT_HOMED THEN
        iOUT_Step := ST120_Pnp_e.Init_HorizontalsToTrack;
    END_IF

ST120_Pnp_e.Init_HorizontalsToTrack:
    IF fb_PnpHorAxis.MoveTo(ST120_PnpHorPos_e.GS).xOUT_InPos THEN
        iOUT_Step := ST120_Pnp_e.Init_adjust_left_clamp;
    END_IF

ST120_Pnp_e.Init_adjust_left_clamp:
    // a piece is in the griper when there is no GS signal
    IF _20_AUTO.recipe.st120.xUseVerLeft THEN
        iOUT_Step := ST120_Pnp_e.Init_adjust_right_clamp;
    ELSE
        iOUT_Step := ST120_Pnp_e.Init_open_left_clamp;
    END_IF

ST120_Pnp_e.Init_open_left_clamp:
    IF fb_gripperLeft.xIN_AS THEN
        IF _20_AUTO.recipe.st120.xUseVerRight THEN
            iOUT_Step := ST120_Pnp_e.Init_adjust_right_clamp;
        ELSE
            iOUT_Step := ST120_Pnp_e.Init_check_if_pces_handled;
        END_IF
    END_IF

ST120_Pnp_e.Init_adjust_right_clamp:
    // a piece is in the griper when there is no GS signal
    IF _20_AUTO.recipe.st120.xUseVerRight THEN
        iOUT_Step := ST120_Pnp_e.Init_check_if_pces_handled;
    ELSE
        iOUT_Step := ST120_Pnp_e.Init_open_right_clamp;
    END_IF

ST120_Pnp_e.Init_open_right_clamp:
    IF fb_gripperRight.xIN_AS THEN
        iOUT_Step := ST120_Pnp_e.Init_check_if_pces_handled;
    END_IF

ST120_Pnp_e.Init_check_if_pces_handled:
    IF (NOT _20_AUTO.recipe.st120.xUseVerLeft AND NOT fb_gripperLeft.xIN_AS) OR
       (NOT _20_AUTO.recipe.st120.xUseVerRight AND NOT fb_gripperRight.xIN_AS) THEN
        bOUT_Error := ST120_Alarm_e.Piece_in_unused_griper;
        iOUT_Step  := ST120_Pnp_e.ERROR;

    ELSIF (_20_AUTO.recipe.st120.xUseVerLeft AND fb_gripperLeft.xOUT_inAS) AND
          (_20_AUTO.recipe.st120.xUseVerRight AND NOT fb_gripperRight.xOUT_inAS) THEN
        bOUT_Error := ST120_Alarm_e.Piece_missing_left_griper;
        iOUT_Step  := ST120_Pnp_e.ERROR;

    ELSIF (_20_AUTO.recipe.st120.xUseVerLeft AND NOT fb_gripperLeft.xOUT_inAS) AND
          (_20_AUTO.recipe.st120.xUseVerRight AND fb_gripperRight.xOUT_inAS) THEN
        bOUT_Error := ST120_Alarm_e.Piece_missing_right_griper;
        iOUT_Step  := ST120_Pnp_e.ERROR;

        // if both are open, we don't make further checks	
		//open meens empty -> get pieces
    ELSIF (NOT _20_AUTO.recipe.st120.xUseVerLeft OR fb_gripperLeft.xOUT_inAS) AND
          (NOT _20_AUTO.recipe.st120.xUseVerRight OR fb_gripperRight.xOUT_inAS) THEN
        iOUT_Step := ST120_Pnp_e.READY;
    ELSE
        iOUT_Step := ST120_Pnp_e.waitOnMover;
    END_IF

(***** READY / INIT DONE *****)
ST120_Pnp_e.READY:    (* Start AUTO,END,LEER,STEP *)
    IF xIN_Start THEN //IF rtSTART.Q THEN
        iOUT_Step := ST120_Pnp_e.START;
    END_IF

(***** START  ZYKLISCH *****)
ST120_Pnp_e.START: (*  *)
    IF xIN_NextStep AND pxFG_Freigabe^ THEN
        IF enState.StateLEER = enIN_State THEN
            IF __ISVALIDREF(Mover) THEN
                IF Mover.GetLastStationDone() > 0 THEN
                    iOUT_Step := ST120_Pnp_e.PnP_Hor_ToRotTablePos;
                ELSE
                    iOUT_Step := ST120_Pnp_e.waitOnMover;
                END_IF
            END_IF
        ELSE
            iOUT_Step := ST120_Pnp_e.PnP_Hor_ToRotTablePos;
        END_IF
    END_IF;

ST120_Pnp_e.PnP_Hor_ToRotTablePos:
    IF xIN_NextStep AND fb_PnpHorAxis.MoveTo(ST120_PnpHorPos_e.AS).xOUT_InPos THEN
        iOUT_Step := ST120_Pnp_e.PnP_WaitOnFeeder;
    END_IF

ST120_Pnp_e.PnP_WaitOnFeeder:
    IF xIN_PceReadyToPick THEN
        iOUT_Step := ST120_Pnp_e.PnP_Ver_RotTableDown;
    END_IF

ST120_Pnp_e.PnP_Ver_RotTableDown:
    IF xIN_NextStep AND fb_PnpVerAxis.MoveTo(ST120_PnpVerPos_e.DownEmpty).xOUT_InPos THEN
        iOUT_Step := ST120_Pnp_e.Gripper_close;
    END_IF;

ST120_Pnp_e.Gripper_close:
    IF xIN_NextStep AND
       (NOT _20_AUTO.recipe.st120.xUseVerLeft OR fb_gripperLeft.xOUT_inGS) AND
       (NOT _20_AUTO.recipe.st120.xUseVerRight OR fb_gripperRight.xOUT_inGS) THEN
        iOUT_Step := ST120_Pnp_e.PnP_Ver_RotTableUp;
    END_IF;

ST120_Pnp_e.PnP_Ver_RotTableUp:
    IF xIN_NextStep AND fb_PnpVerAxis.MoveTo(ST120_PnpVerPos_e.UpFull).xOUT_InPos THEN
        iOUT_Step := ST120_Pnp_e.PnP_Hor_ToTrackPos;
    END_IF;

ST120_Pnp_e.PnP_Hor_ToTrackPos:
    IF xIN_NextStep AND fb_PnpHorAxis.MoveTo(ST120_PnpHorPos_e.GS).xOUT_InPos THEN
        iOUT_Step := ST120_Pnp_e.waitOnMover;
    END_IF

ST120_Pnp_e.waitOnMover: (*  *)
    IF xIN_NextStep AND __ISVALIDREF(Mover) OR HMI.bArForceCyclusState[StationList_e.ST120] THEN
        IF Mover.GetLastStationDone() >= INT#120 THEN
            iOUT_Step := ST120_Pnp_e.SYNC_MOVER_LEAVE;
        ELSIF Mover.GetLastStationDone() < INT#105 THEN
            iOUT_Step := ST120_Pnp_e.SYNC_MOVER_LEAVE;
        ELSE
            iOUT_Step := ST120_Pnp_e.PnP_Ver_ShuttleDown;
        END_IF
    END_IF;

ST120_Pnp_e.PnP_Ver_ShuttleDown:
    IF xIN_NextStep AND fb_PnpVerAxis.MoveTo(ST120_PnpVerPos_e.DownFullQuick).xOUT_InPos THEN
        iOUT_Step := ST120_Pnp_e.PnP_Ver_ShuttleTorqueControl;

        IF __ISVALIDREF(Mover) THEN
            IF NOT Mover.SetLastStation(120) THEN
                ASSERT(0);
            END_IF
        END_IF
    END_IF;

// We need a fb that enables for us torque control. Here we just go a bit further
ST120_Pnp_e.PnP_Ver_ShuttleTorqueControl:
    IF xIN_NextStep AND fb_PnpVerAxis.MoveTo(ST120_PnpVerPos_e.DownFullTorqueControl).xOUT_InPos THEN
        iOUT_Step := ST120_Pnp_e.Gripper_open;
    END_IF;

ST120_Pnp_e.Gripper_open:
    IF xIN_NextStep AND
       (NOT _20_AUTO.recipe.st120.xUseVerLeft OR fb_gripperLeft.xOUT_inAS) AND
       (NOT _20_AUTO.recipe.st120.xUseVerRight OR fb_gripperRight.xOUT_inAS) THEN
        iOUT_Step := ST120_Pnp_e.PnP_Ver_ShuttleUp;
    END_IF;

ST120_Pnp_e.PnP_Ver_ShuttleUp:
    IF xIN_NextStep AND fb_PnpVerAxis.MoveTo(ST120_PnpVerPos_e.UpEmpty).xOUT_InPos THEN
        iOUT_Step := ST120_Pnp_e.SYNC_MOVER_LEAVE;

        IF __ISVALIDREF(Mover) THEN
            IF NOT Mover.SetLastStation(120) THEN
                ASSERT(0);
            END_IF
        END_IF
    END_IF;

ST120_Pnp_e.SYNC_MOVER_LEAVE:
    // The mover needs to be taken by MoverMan
    IF NOT __ISVALIDREF(Mover) THEN
        IF (NOT _20_AUTO.recipe.st120.xUseVerLeft OR fb_gripperLeft.xOUT_inAS) AND
           (NOT _20_AUTO.recipe.st120.xUseVerRight OR fb_gripperRight.xOUT_inAS) THEN
            iOUT_Step := ST120_Pnp_e.DONE;
        ELSE
            iOUT_Step := ST120_Pnp_e.waitOnMover;
        END_IF
    END_IF

(***** DONE *****)
ST120_Pnp_e.DONE: (* Letzter Schritt  *)
    IF NOT xIN_AlarmAktiv THEN
        //AUTO
        IF (enIN_State = StateAUTO) AND xIN_RestartCYCL THEN
            iOUT_Step := ST120_Pnp_e.START;
            //STEP / END / LEERFAHREN restart
        ELSIF (enIN_State < StateAUTO) AND (enIN_State >= enState.StateSTEP) AND xIN_RestartCYCL THEN
            iOUT_Step := ST120_Pnp_e.START;
            //STEP / END / LEERFAHREN fertig
        ELSIF (enIN_State = StateREADY) THEN
            iOUT_Step := ST120_Pnp_e.READY;
        END_IF;
    END_IF;

(************ ERROR *************)
ST120_Pnp_e.ERROR: (* ERROR *) ;

END_CASE;

END_FUNCTION_BLOCK

// ---- POUs/20_AUTO/ST120/POU_ALARM_120.TcPOU
PROGRAM POU_ALARM_120
VAR_INPUT
    xIN_QUIT      : BOOL; // Alarm quittieren
    iIN_ArraySize : INT;
    pstrIN_ALARM  : POINTER TO structAlarm;       // Array Alarmstruktur
    refPOU        : REFERENCE TO FB_AUT_ABSTRACT; // the POU to test
END_VAR
VAR_OUTPUT
    xOUT_AL_ST : BOOL; // Alarm Station aktiv
END_VAR
VAR
    //Alarmbaustein
    _FB_ALARM_ST : FB_ALARM;
    //Local
    iIndex : INT; // Index For Schleife	
END_VAR
VAR CONSTANT
    sDefString : STRING := 'Error ST120,'; // Station #
END_VAR

(********************** INITIALISIERE VARIABLEN ****************************)
FOR iIndex := 0 TO iIN_ArraySize - 1 DO
    pstrIN_ALARM[iIndex].xAlarmIN   := FALSE;
    pstrIN_ALARM[iIndex].xAlarmOFF  := FALSE;
    pstrIN_ALARM[iIndex].xAlarmSAVE := TRUE;
    pstrIN_ALARM[iIndex].xAlarmQUIT := xIN_QUIT;
    pstrIN_ALARM[iIndex].tAlarmVERZ := T#100MS;
    pstrIN_ALARM[iIndex].sAlarmText := '';
    pstrIN_ALARM[iIndex].bAlarmNr   := 0;
END_FOR

(********************** ALARME ****************************)
pstrIN_ALARM[0].xAlarmIN   := (refPOU.bOUT_ErrorNum = ST120_Alarm_e.Axis_120_01Y_error);
pstrIN_ALARM[0].sAlarmText := CONCAT(sDefString, ' Axis 01Y in error');
pstrIN_ALARM[0].bAlarmNr   := 0;

pstrIN_ALARM[1].xAlarmIN   := (refPOU.bOUT_ErrorNum = ST120_Alarm_e.Axis_120_02Z_error);
pstrIN_ALARM[1].sAlarmText := CONCAT(sDefString, ' Axis 02Z in error');
pstrIN_ALARM[1].bAlarmNr   := 0;

pstrIN_ALARM[2].xAlarmIN   := (refPOU.bOUT_ErrorNum = ST120_Alarm_e.Cylinder_griper_left);
pstrIN_ALARM[2].sAlarmText := CONCAT(sDefString, ' Cylinder .05 gripper right');
pstrIN_ALARM[2].bAlarmNr   := 0;

pstrIN_ALARM[3].xAlarmIN   := (refPOU.bOUT_ErrorNum = ST120_Alarm_e.Cylinder_griper_right);
pstrIN_ALARM[3].sAlarmText := CONCAT(sDefString, ' Cylinder .06 gripper left');
pstrIN_ALARM[3].bAlarmNr   := 0;

pstrIN_ALARM[4].xAlarmIN   := (refPOU.bOUT_ErrorNum = ST120_Alarm_e.Cylinder_pivot_left);
pstrIN_ALARM[4].sAlarmText := CONCAT(sDefString, ' Cylinder .06 pivot left');
pstrIN_ALARM[4].bAlarmNr   := 0;

pstrIN_ALARM[5].xAlarmIN   := (refPOU.bOUT_ErrorNum = ST120_Alarm_e.Cylinder_pivot_right);
pstrIN_ALARM[5].sAlarmText := CONCAT(sDefString, ' Cylinder .06 pivot left');
pstrIN_ALARM[5].bAlarmNr   := 0;

pstrIN_ALARM[6].xAlarmIN   := (refPOU.bOUT_ErrorNum = ST120_Alarm_e.Cylinder_hublader_left);
pstrIN_ALARM[6].sAlarmText := CONCAT(sDefString, ' Cylinder .06 hublader left');
pstrIN_ALARM[6].bAlarmNr   := 0;

pstrIN_ALARM[7].xAlarmIN   := (refPOU.bOUT_ErrorNum = ST120_Alarm_e.Cylinder_hublader_right);
pstrIN_ALARM[7].sAlarmText := CONCAT(sDefString, ' Cylinder .06 hublader left');
pstrIN_ALARM[7].bAlarmNr   := 0;

pstrIN_ALARM[8].xAlarmIN   := (refPOU.bOUT_ErrorNum = ST120_Alarm_e.Piece_in_unused_griper);
pstrIN_ALARM[8].sAlarmText := CONCAT(sDefString, ' One part is handled by a unused griper');
pstrIN_ALARM[8].bAlarmNr   := 0;

pstrIN_ALARM[9].xAlarmIN   := (refPOU.bOUT_ErrorNum = ST120_Alarm_e.Piece_missing_left_griper);
pstrIN_ALARM[9].sAlarmText := CONCAT(sDefString, ' A piece is missing in the left griper');
pstrIN_ALARM[9].bAlarmNr   := 0;

pstrIN_ALARM[10].xAlarmIN   := (refPOU.bOUT_ErrorNum = ST120_Alarm_e.Piece_missing_right_griper);
pstrIN_ALARM[10].sAlarmText := CONCAT(sDefString, ' A piece is missing in the right griper');
pstrIN_ALARM[10].bAlarmNr   := 0;

pstrIN_ALARM[11].xAlarmIN   := (refPOU.bOUT_ErrorNum = ST120_Alarm_e.Feeder_empty);
pstrIN_ALARM[11].sAlarmText := CONCAT(sDefString, ' The feeder is empty');
pstrIN_ALARM[11].bAlarmNr   := 0;

pstrIN_ALARM[12].xAlarmIN   := (refPOU.bOUT_ErrorNum = ST120_Alarm_e.Feeder_error);
pstrIN_ALARM[12].sAlarmText := CONCAT(sDefString, ' One part of the feeder is in error');
pstrIN_ALARM[12].bAlarmNr   := 0;

pstrIN_ALARM[13].xAlarmIN   := (refPOU.bOUT_ErrorNum = ST120_Alarm_e.Piece_in_unused_pivot);
pstrIN_ALARM[13].sAlarmText := CONCAT(sDefString, ' One part is handled by a unused pivot');
pstrIN_ALARM[13].bAlarmNr   := 0;

pstrIN_ALARM[14].xAlarmIN   := (refPOU.bOUT_ErrorNum = ST120_Alarm_e.Piece_missing_left_pivot);
pstrIN_ALARM[14].sAlarmText := CONCAT(sDefString, ' A piece is missing in the left pivot');
pstrIN_ALARM[14].bAlarmNr   := 0;

pstrIN_ALARM[15].xAlarmIN   := (refPOU.bOUT_ErrorNum = ST120_Alarm_e.Piece_missing_right_pivor);
pstrIN_ALARM[15].sAlarmText := CONCAT(sDefString, ' A piece is missing in the right pivot');
pstrIN_ALARM[15].bAlarmNr   := 0;

(********************** ALARM FB ****************************)
_FB_ALARM_ST(pstrIN_Alarm  := pstrIN_ALARM,
             iIN_ArraySize := ST120_Alarm_e._max);

(********************** ALARM FB ****************************)
xOUT_AL_ST := FALSE;

FOR iIndex := 0 TO iIN_ArraySize - 1 DO
    IF pstrIN_ALARM[iIndex].xAlarmOUT THEN
        xOUT_AL_ST := TRUE;
    END_IF
END_FOR

END_PROGRAM

